LIN {X 0.001,Y -352.403,Z 1885.595,A 0.000,B 0.000,C 90.000,E1 287.166} C_DIS
LIN {X -0.016,Y -356.539,Z 1885.590,A 0.000,B 0.000,C 90.000,E1 286.260} C_DIS
LIN {X -0.091,Y -360.124,Z 1885.585,A 0.000,B 0.000,C 90.000,E1 285.371} C_DIS
LIN {X -0.135,Y -363.075,Z 1885.580,A 0.000,B 0.000,C 90.000,E1 284.481} C_DIS
LIN {X -0.125,Y -364.654,Z 1885.577,A 0.000,B 0.000,C 90.000,E1 283.883} C_DIS
LIN {X -0.190,Y -365.903,Z 1885.574,A 0.000,B 0.000,C 90.000,E1 283.300} C_DIS
LIN {X 0.194,Y -366.725,Z 1885.570,A 0.000,B 0.000,C 90.000,E1 282.647} C_DIS
LIN {X 0.148,Y -367.195,Z 1885.567,A 0.000,B 0.000,C 90.000,E1 282.063} C_DIS
LIN {X 0.107,Y -367.233,Z 1885.564,A 0.000,B 0.000,C 90.000,E1 281.478} C_DIS
LIN {X 0.069,Y -366.898,Z 1885.561,A 0.000,B 0.000,C 90.000,E1 280.894} C_DIS
LIN {X 0.032,Y -366.222,Z 1885.557,A 0.000,B 0.000,C 90.000,E1 280.310} C_DIS
LIN {X -0.009,Y -365.133,Z 1885.554,A 0.000,B 0.000,C 90.000,E1 279.726} C_DIS
LIN {X -0.115,Y -363.688,Z 1885.551,A 0.000,B 0.000,C 90.000,E1 279.151} C_DIS
LIN {X -0.167,Y -361.942,Z 1885.547,A 0.000,B 0.000,C 90.000,E1 278.568} C_DIS
LIN {X 0.040,Y -358.752,Z 1885.542,A 0.000,B 0.000,C 90.000,E1 277.644} C_DIS
LIN {X -0.139,Y -354.719,Z 1885.537,A 0.000,B 0.000,C 90.000,E1 276.777} C_DIS
LIN {X 0.059,Y -351.476,Z 1885.534,A 0.000,B 0.000,C 90.000,E1 276.144} C_DIS
LIN {X -0.111,Y -347.742,Z 1885.531,A 0.000,B 0.000,C 90.000,E1 275.568} C_DIS
LIN {X 0.045,Y -343.441,Z 1885.527,A 0.000,B 0.000,C 90.000,E1 274.935} C_DIS
LIN {X -0.165,Y -338.448,Z 1885.524,A 0.000,B 0.000,C 90.000,E1 274.359} C_DIS
LIN {X -0.059,Y -332.829,Z 1885.521,A 0.000,B 0.000,C 90.000,E1 273.726} C_DIS
LIN {X -0.066,Y -326.939,Z 1885.517,A 0.000,B 0.000,C 90.000,E1 273.154} C_DIS
LIN {X 0.124,Y -320.558,Z 1885.514,A 0.000,B 0.000,C 90.000,E1 272.579} C_DIS
LIN {X 0.017,Y -314.110,Z 1885.512,A 0.000,B 0.000,C 90.000,E1 272.121} C_DIS
LIN {X -0.084,Y -307.356,Z 1885.509,A 0.000,B 0.000,C 90.000,E1 271.718} C_DIS
LIN {X -0.136,Y -300.498,Z 1885.507,A 0.000,B 0.000,C 90.000,E1 271.375} C_DIS
LIN {X 0.073,Y -292.946,Z 1885.506,A 0.000,B 0.000,C 90.000,E1 271.031} C_DIS
LIN {X 0.051,Y -285.090,Z 1885.505,A 0.000,B 0.000,C 90.000,E1 270.802} C_DIS
LIN {X -0.071,Y -273.586,Z 1885.503,A 0.000,B 0.000,C 90.000,E1 270.573} C_DIS
LIN {X 0.101,Y -252.260,Z 1885.501,A 0.000,B 0.000,C 90.000,E1 270.115} C_DIS
LIN {X -0.047,Y -240.338,Z 1885.500,A 0.000,B 0.000,C 90.000,E1 269.943} C_DIS
LIN {X -0.106,Y -228.165,Z 1885.499,A 0.000,B 0.000,C 90.000,E1 269.828} C_DIS
LIN {X 0.098,Y -226.995,Z 1885.499,A 0.000,B 0.000,C 90.000,E1 269.771} C_DIS
LIN {X 0.059,Y -181.515,Z 1885.499,A 0.000,B 0.000,C 90.000,E1 269.771} C_DIS
LIN {X 0.072,Y -180.907,Z 1885.475,A 0.000,B 0.000,C 90.000,E1 265.469} C_DIS
LIN {X -0.050,Y -180.746,Z 1885.470,A 0.000,B 0.000,C 90.000,E1 264.666} C_DIS
LIN {X 0.017,Y -178.838,Z 1885.442,A 0.000,B 0.000,C 90.000,E1 259.577} C_DIS
LIN {X -0.085,Y -175.882,Z 1885.414,A 0.000,B 0.000,C 90.000,E1 254.519} C_DIS
LIN {X 0.021,Y -174.545,Z 1885.404,A 0.000,B 0.000,C 90.000,E1 252.779} C_DIS
LIN {X -0.046,Y -171.530,Z 1885.381,A 0.000,B 0.000,C 90.000,E1 248.518} C_DIS
LIN {X -0.053,Y -167.755,Z 1885.357,A 0.000,B 0.000,C 90.000,E1 244.204} C_DIS
LIN {X 0.037,Y -166.460,Z 1885.347,A 0.000,B 0.000,C 90.000,E1 242.436} C_DIS
LIN {X 0.026,Y -163.175,Z 1885.328,A 0.000,B 0.000,C 90.000,E1 238.948} C_DIS
LIN {X 0.075,Y -161.135,Z 1885.313,A 0.000,B 0.000,C 90.000,E1 236.294} C_DIS
LIN {X -0.023,Y -157.156,Z 1885.288,A 0.000,B 0.000,C 90.000,E1 231.904} C_DIS
LIN {X 0.001,Y -155.888,Z 1885.278,A 0.000,B 0.000,C 90.000,E1 230.114} C_DIS
LIN {X -0.041,Y -152.138,Z 1885.254,A 0.000,B 0.000,C 90.000,E1 225.648} C_DIS
LIN {X -0.021,Y -150.388,Z 1885.239,A 0.000,B 0.000,C 90.000,E1 222.933} C_DIS
LIN {X 0.003,Y -147.119,Z 1885.213,A 0.000,B 0.000,C 90.000,E1 218.382} C_DIS
LIN {X -0.005,Y -145.684,Z 1885.198,A 0.000,B 0.000,C 90.000,E1 215.644} C_DIS
LIN {X -0.008,Y -143.065,Z 1885.172,A 0.000,B 0.000,C 90.000,E1 211.052} C_DIS
LIN {X 0.050,Y -141.687,Z 1885.152,A 0.000,B 0.000,C 90.000,E1 207.334} C_DIS
LIN {X -0.022,Y -139.459,Z 1885.116,A 0.000,B 0.000,C 90.000,E1 200.865} C_DIS
LIN {X 0.079,Y -139.194,Z 1885.105,A 0.000,B 0.000,C 90.000,E1 198.960} C_DIS
LIN {X -0.035,Y -138.324,Z 1885.054,A 0.000,B 0.000,C 90.000,E1 189.670} C_DIS
LIN {X -0.030,Y -139.452,Z 1885.007,A 0.000,B 0.000,C 90.000,E1 181.260} C_DIS
LIN {X 0.050,Y -140.998,Z 1884.976,A 0.000,B 0.000,C 90.000,E1 175.641} C_DIS
LIN {X -0.001,Y -142.753,Z 1884.955,A 0.000,B 0.000,C 90.000,E1 171.951} C_DIS
LIN {X -0.044,Y -145.153,Z 1884.930,A 0.000,B 0.000,C 90.000,E1 167.353} C_DIS
LIN {X -0.052,Y -147.776,Z 1884.909,A 0.000,B 0.000,C 90.000,E1 163.685} C_DIS
LIN {X 0.028,Y -150.453,Z 1884.889,A 0.000,B 0.000,C 90.000,E1 160.007} C_DIS
LIN {X -0.038,Y -153.902,Z 1884.869,A 0.000,B 0.000,C 90.000,E1 156.410} C_DIS
LIN {X 0.028,Y -157.313,Z 1884.849,A 0.000,B 0.000,C 90.000,E1 152.794} C_DIS
LIN {X -0.026,Y -161.500,Z 1884.829,A 0.000,B 0.000,C 90.000,E1 149.253} C_DIS
LIN {X -0.010,Y -165.699,Z 1884.810,A 0.000,B 0.000,C 90.000,E1 145.722} C_DIS
LIN {X 0.116,Y -170.643,Z 1884.790,A 0.000,B 0.000,C 90.000,E1 142.190} C_DIS
LIN {X 0.028,Y -175.519,Z 1884.771,A 0.000,B 0.000,C 90.000,E1 138.771} C_DIS
LIN {X 0.023,Y -181.139,Z 1884.752,A 0.000,B 0.000,C 90.000,E1 135.364} C_DIS
LIN {X 0.021,Y -186.590,Z 1884.733,A 0.000,B 0.000,C 90.000,E1 132.000} C_DIS
LIN {X 0.091,Y -191.201,Z 1884.719,A 0.000,B 0.000,C 90.000,E1 129.483} C_DIS
LIN {X 0.015,Y -197.011,Z 1884.701,A 0.000,B 0.000,C 90.000,E1 126.217} C_DIS
LIN {X -0.066,Y -200.281,Z 1884.692,A 0.000,B 0.000,C 90.000,E1 124.612} C_DIS
LIN {X -0.073,Y -207.773,Z 1884.670,A 0.000,B 0.000,C 90.000,E1 120.590} C_DIS
LIN {X 0.113,Y -210.945,Z 1884.661,A 0.000,B 0.000,C 90.000,E1 118.949} C_DIS
LIN {X -0.066,Y -216.817,Z 1884.644,A 0.000,B 0.000,C 90.000,E1 115.848} C_DIS
LIN {X 0.083,Y -218.433,Z 1884.639,A 0.000,B 0.000,C 90.000,E1 115.027} C_DIS
LIN {X -0.079,Y -221.158,Z 1884.630,A 0.000,B 0.000,C 90.000,E1 113.515} C_DIS
LIN {X -0.007,Y -224.115,Z 1884.621,A 0.000,B 0.000,C 90.000,E1 111.844} C_DIS
LIN {X -0.044,Y -283.396,Z 1884.621,A 0.000,B 0.000,C 90.000,E1 111.844} C_DIS
LIN {X 0.060,Y -286.175,Z 1884.621,A 0.000,B 0.000,C 90.000,E1 111.770} C_DIS
LIN {X 0.099,Y -291.202,Z 1884.619,A 0.000,B 0.000,C 90.000,E1 111.461} C_DIS
LIN {X 0.032,Y -293.997,Z 1884.618,A 0.000,B 0.000,C 90.000,E1 111.173} C_DIS
LIN {X 0.068,Y -296.048,Z 1884.616,A 0.000,B 0.000,C 90.000,E1 110.865} C_DIS
LIN {X -0.046,Y -309.093,Z 1884.603,A 0.000,B 0.000,C 90.000,E1 108.598} C_DIS
LIN {X 0.047,Y -323.638,Z 1884.591,A 0.000,B 0.000,C 90.000,E1 106.315} C_DIS
LIN {X 0.008,Y -337.287,Z 1884.580,A 0.000,B 0.000,C 90.000,E1 104.426} C_DIS
LIN {X -0.102,Y -352.119,Z 1884.570,A 0.000,B 0.000,C 90.000,E1 102.591} C_DIS
LIN {X -0.120,Y -370.511,Z 1884.558,A 0.000,B 0.000,C 90.000,E1 100.546} C_DIS
LIN {X -0.077,Y -389.326,Z 1884.548,A 0.000,B 0.000,C 90.000,E1 98.681} C_DIS
LIN {X 0.195,Y -408.561,Z 1884.539,A 0.000,B 0.000,C 90.000,E1 96.947} C_DIS
LIN {X -0.005,Y -430.922,Z 1884.529,A 0.000,B 0.000,C 90.000,E1 95.220} C_DIS
LIN {X 0.152,Y -439.357,Z 1884.526,A 0.000,B 0.000,C 90.000,E1 94.588} C_DIS
LIN {X -0.073,Y -441.584,Z 1884.525,A 0.000,B 0.000,C 90.000,E1 94.416} C_DIS
LIN {X -0.138,Y -443.567,Z 1884.523,A 0.000,B 0.000,C 90.000,E1 94.188} C_DIS
LIN {X -0.172,Y -445.091,Z 1884.522,A 0.000,B 0.000,C 90.000,E1 93.955} C_DIS
LIN {X 0.007,Y -446.387,Z 1884.520,A 0.000,B 0.000,C 90.000,E1 93.669} C_DIS
LIN {X 0.188,Y -447.352,Z 1884.519,A 0.000,B 0.000,C 90.000,E1 93.383} C_DIS
LIN {X 0.146,Y -448.456,Z 1884.516,A 0.000,B 0.000,C 90.000,E1 92.865} C_DIS
LIN {X 0.086,Y -448.602,Z 1884.513,A 0.000,B 0.000,C 90.000,E1 92.350} C_DIS
LIN {X 0.037,Y -447.816,Z 1884.510,A 0.000,B 0.000,C 90.000,E1 91.835} C_DIS
LIN {X 0.000,Y -445.975,Z 1884.507,A 0.000,B 0.000,C 90.000,E1 91.318} C_DIS
LIN {X -0.053,Y -442.903,Z 1884.504,A 0.000,B 0.000,C 90.000,E1 90.802} C_DIS
LIN {X -0.162,Y -431.386,Z 1884.494,A 0.000,B 0.000,C 90.000,E1 88.969} C_DIS
LIN {X -0.184,Y -421.317,Z 1884.485,A 0.000,B 0.000,C 90.000,E1 87.364} C_DIS
LIN {X 0.139,Y -409.543,Z 1884.475,A 0.000,B 0.000,C 90.000,E1 85.412} C_DIS
LIN {X -0.166,Y -397.645,Z 1884.464,A 0.000,B 0.000,C 90.000,E1 83.514} C_DIS
LIN {X 0.167,Y -385.682,Z 1884.453,A 0.000,B 0.000,C 90.000,E1 81.489} C_DIS
LIN {X -0.072,Y -373.809,Z 1884.442,A 0.000,B 0.000,C 90.000,E1 79.511} C_DIS
LIN {X 0.188,Y -355.793,Z 1884.424,A 0.000,B 0.000,C 90.000,E1 76.228} C_DIS
LIN {X -0.142,Y -341.985,Z 1884.409,A 0.000,B 0.000,C 90.000,E1 73.559} C_DIS
LIN {X 0.129,Y -330.104,Z 1884.395,A 0.000,B 0.000,C 90.000,E1 71.040} C_DIS
LIN {X -0.057,Y -317.077,Z 1884.379,A 0.000,B 0.000,C 90.000,E1 68.230} C_DIS
LIN {X 0.046,Y -304.672,Z 1884.363,A 0.000,B 0.000,C 90.000,E1 65.305} C_DIS
LIN {X 0.048,Y -295.143,Z 1884.350,A 0.000,B 0.000,C 90.000,E1 62.999} C_DIS
LIN {X -0.020,Y -285.826,Z 1884.337,A 0.000,B 0.000,C 90.000,E1 60.667} C_DIS
LIN {X -0.010,Y -276.398,Z 1884.324,A 0.000,B 0.000,C 90.000,E1 58.280} C_DIS
LIN {X -0.150,Y -266.915,Z 1884.310,A 0.000,B 0.000,C 90.000,E1 55.881} C_DIS
LIN {X 0.025,Y -257.306,Z 1884.297,A 0.000,B 0.000,C 90.000,E1 53.371} C_DIS
LIN {X -0.120,Y -247.700,Z 1884.283,A 0.000,B 0.000,C 90.000,E1 50.884} C_DIS
LIN {X -0.146,Y -238.217,Z 1884.268,A 0.000,B 0.000,C 90.000,E1 48.324} C_DIS
LIN {X -0.021,Y -226.401,Z 1884.250,A 0.000,B 0.000,C 90.000,E1 44.919} C_DIS
LIN {X -0.055,Y -215.186,Z 1884.230,A 0.000,B 0.000,C 90.000,E1 41.472} C_DIS
LIN {X 0.051,Y -205.981,Z 1884.213,A 0.000,B 0.000,C 90.000,E1 38.302} C_DIS
LIN {X 0.048,Y -197.685,Z 1884.195,A 0.000,B 0.000,C 90.000,E1 35.105} C_DIS
LIN {X -0.042,Y -190.108,Z 1884.177,A 0.000,B 0.000,C 90.000,E1 31.878} C_DIS
LIN {X -0.025,Y -183.281,Z 1884.159,A 0.000,B 0.000,C 90.000,E1 28.565} C_DIS
LIN {X -0.031,Y -177.125,Z 1884.140,A 0.000,B 0.000,C 90.000,E1 25.207} C_DIS
LIN {X 0.063,Y -171.807,Z 1884.121,A 0.000,B 0.000,C 90.000,E1 21.770} C_DIS
LIN {X -0.061,Y -167.257,Z 1884.102,A 0.000,B 0.000,C 90.000,E1 18.362} C_DIS
LIN {X 0.082,Y -163.533,Z 1884.083,A 0.000,B 0.000,C 90.000,E1 14.828} C_DIS
LIN {X -0.087,Y -159.741,Z 1884.058,A 0.000,B 0.000,C 90.000,E1 10.489} C_DIS
LIN {X -0.023,Y -157.111,Z 1884.033,A 0.000,B 0.000,C 90.000,E1 6.030} C_DIS
LIN {X 0.000,Y -154.819,Z 1884.000,A 0.000,B 0.000,C 90.000,E1 360.000} C_DIS
LIN {X -0.016,Y -154.068,Z 1883.948,A 0.000,B 0.000,C 90.000,E1 350.557} C_DIS
LIN {X -0.014,Y -156.089,Z 1883.908,A 0.000,B 0.000,C 90.000,E1 343.378} C_DIS
LIN {X 0.017,Y -158.516,Z 1883.883,A 0.000,B 0.000,C 90.000,E1 338.901} C_DIS
LIN {X 0.031,Y -162.145,Z 1883.858,A 0.000,B 0.000,C 90.000,E1 334.460} C_DIS
LIN {X 0.082,Y -166.114,Z 1883.839,A 0.000,B 0.000,C 90.000,E1 330.923} C_DIS
LIN {X 0.014,Y -169.717,Z 1883.824,A 0.000,B 0.000,C 90.000,E1 328.329} C_DIS
LIN {X 0.051,Y -173.031,Z 1883.812,A 0.000,B 0.000,C 90.000,E1 326.215} C_DIS
LIN {X 0.035,Y -182.366,Z 1883.812,A 0.000,B 0.000,C 90.000,E1 326.215} C_DIS
LIN {X 0.053,Y -185.804,Z 1883.810,A 0.000,B 0.000,C 90.000,E1 325.722} C_DIS
LIN {X 0.055,Y -188.638,Z 1883.805,A 0.000,B 0.000,C 90.000,E1 324.895} C_DIS
LIN {X 0.040,Y -190.835,Z 1883.800,A 0.000,B 0.000,C 90.000,E1 324.069} C_DIS
LIN {X -0.001,Y -194.525,Z 1883.791,A 0.000,B 0.000,C 90.000,E1 322.431} C_DIS
LIN {X -0.036,Y -199.322,Z 1883.778,A 0.000,B 0.000,C 90.000,E1 319.989} C_DIS
LIN {X -0.086,Y -206.996,Z 1883.755,A 0.000,B 0.000,C 90.000,E1 315.972} C_DIS
LIN {X 0.014,Y -210.390,Z 1883.746,A 0.000,B 0.000,C 90.000,E1 314.352} C_DIS
LIN {X 0.054,Y -215.246,Z 1883.735,A 0.000,B 0.000,C 90.000,E1 312.366} C_DIS
LIN {X -0.029,Y -219.816,Z 1883.727,A 0.000,B 0.000,C 90.000,E1 310.825} C_DIS
LIN {X -0.028,Y -225.338,Z 1883.718,A 0.000,B 0.000,C 90.000,E1 309.277} C_DIS
LIN {X -0.008,Y -233.096,Z 1883.708,A 0.000,B 0.000,C 90.000,E1 307.363} C_DIS
LIN {X -0.148,Y -246.896,Z 1883.691,A 0.000,B 0.000,C 90.000,E1 304.405} C_DIS
LIN {X -0.004,Y -256.206,Z 1883.681,A 0.000,B 0.000,C 90.000,E1 302.546} C_DIS
LIN {X 0.129,Y -272.970,Z 1883.665,A 0.000,B 0.000,C 90.000,E1 299.667} C_DIS
LIN {X 0.053,Y -290.803,Z 1883.650,A 0.000,B 0.000,C 90.000,E1 296.924} C_DIS
LIN {X 0.128,Y -304.184,Z 1883.638,A 0.000,B 0.000,C 90.000,E1 294.899} C_DIS
LIN {X 0.139,Y -315.278,Z 1883.629,A 0.000,B 0.000,C 90.000,E1 293.259} C_DIS
LIN {X 0.084,Y -326.017,Z 1883.620,A 0.000,B 0.000,C 90.000,E1 291.663} C_DIS
LIN {X -0.088,Y -334.306,Z 1883.613,A 0.000,B 0.000,C 90.000,E1 290.429} C_DIS
LIN {X 0.162,Y -340.187,Z 1883.608,A 0.000,B 0.000,C 90.000,E1 289.450} C_DIS
LIN {X 0.040,Y -345.657,Z 1883.603,A 0.000,B 0.000,C 90.000,E1 288.544} C_DIS
LIN {X -0.039,Y -350.699,Z 1883.598,A 0.000,B 0.000,C 90.000,E1 287.638} C_DIS
LIN {X -0.068,Y -355.164,Z 1883.593,A 0.000,B 0.000,C 90.000,E1 286.732} C_DIS
LIN {X -0.163,Y -358.994,Z 1883.588,A 0.000,B 0.000,C 90.000,E1 285.843} C_DIS
LIN {X 0.177,Y -361.272,Z 1883.585,A 0.000,B 0.000,C 90.000,E1 285.190} C_DIS
LIN {X 0.184,Y -363.238,Z 1883.581,A 0.000,B 0.000,C 90.000,E1 284.592} C_DIS
LIN {X 0.106,Y -364.874,Z 1883.578,A 0.000,B 0.000,C 90.000,E1 284.008} C_DIS
LIN {X 0.129,Y -366.174,Z 1883.575,A 0.000,B 0.000,C 90.000,E1 283.411} C_DIS
LIN {X 0.075,Y -367.127,Z 1883.571,A 0.000,B 0.000,C 90.000,E1 282.827} C_DIS
LIN {X 0.031,Y -367.638,Z 1883.568,A 0.000,B 0.000,C 90.000,E1 282.243} C_DIS
LIN {X -0.006,Y -367.773,Z 1883.565,A 0.000,B 0.000,C 90.000,E1 281.658} C_DIS
LIN {X -0.039,Y -367.520,Z 1883.562,A 0.000,B 0.000,C 90.000,E1 281.074} C_DIS
LIN {X -0.071,Y -366.899,Z 1883.558,A 0.000,B 0.000,C 90.000,E1 280.489} C_DIS
LIN {X -0.107,Y -365.890,Z 1883.555,A 0.000,B 0.000,C 90.000,E1 279.905} C_DIS
LIN {X -0.148,Y -364.512,Z 1883.552,A 0.000,B 0.000,C 90.000,E1 279.321} C_DIS
LIN {X 0.107,Y -362.801,Z 1883.548,A 0.000,B 0.000,C 90.000,E1 278.690} C_DIS
LIN {X 0.015,Y -359.690,Z 1883.543,A 0.000,B 0.000,C 90.000,E1 277.814} C_DIS
LIN {X -0.112,Y -357.204,Z 1883.540,A 0.000,B 0.000,C 90.000,E1 277.239} C_DIS
LIN {X 0.046,Y -352.729,Z 1883.535,A 0.000,B 0.000,C 90.000,E1 276.315} C_DIS
LIN {X -0.119,Y -349.129,Z 1883.532,A 0.000,B 0.000,C 90.000,E1 275.739} C_DIS
LIN {X 0.045,Y -344.915,Z 1883.528,A 0.000,B 0.000,C 90.000,E1 275.106} C_DIS
LIN {X -0.158,Y -340.117,Z 1883.525,A 0.000,B 0.000,C 90.000,E1 274.531} C_DIS
LIN {X -0.050,Y -334.635,Z 1883.522,A 0.000,B 0.000,C 90.000,E1 273.898} C_DIS
LIN {X -0.021,Y -325.851,Z 1883.517,A 0.000,B 0.000,C 90.000,E1 273.037} C_DIS
LIN {X -0.020,Y -319.652,Z 1883.514,A 0.000,B 0.000,C 90.000,E1 272.522} C_DIS
LIN {X -0.061,Y -313.156,Z 1883.511,A 0.000,B 0.000,C 90.000,E1 272.064} C_DIS
LIN {X -0.089,Y -306.393,Z 1883.509,A 0.000,B 0.000,C 90.000,E1 271.661} C_DIS
LIN {X -0.103,Y -299.365,Z 1883.507,A 0.000,B 0.000,C 90.000,E1 271.318} C_DIS
LIN {X -0.102,Y -291.908,Z 1883.506,A 0.000,B 0.000,C 90.000,E1 271.031} C_DIS
LIN {X -0.080,Y -284.020,Z 1883.504,A 0.000,B 0.000,C 90.000,E1 270.802} C_DIS
LIN {X 0.003,Y -268.400,Z 1883.503,A 0.000,B 0.000,C 90.000,E1 270.458} C_DIS
LIN {X -0.028,Y -250.496,Z 1883.501,A 0.000,B 0.000,C 90.000,E1 270.115} C_DIS
LIN {X 0.097,Y -238.266,Z 1883.500,A 0.000,B 0.000,C 90.000,E1 269.885} C_DIS
LIN {X -0.098,Y -227.892,Z 1883.499,A 0.000,B 0.000,C 90.000,E1 269.828} C_DIS
LIN {X 0.101,Y -225.810,Z 1883.499,A 0.000,B 0.000,C 90.000,E1 269.771} C_DIS
LIN {X 0.059,Y -181.515,Z 1883.499,A 0.000,B 0.000,C 90.000,E1 269.771} C_DIS
LIN {X -0.011,Y -180.907,Z 1883.475,A 0.000,B 0.000,C 90.000,E1 265.527} C_DIS
LIN {X 0.046,Y -180.760,Z 1883.470,A 0.000,B 0.000,C 90.000,E1 264.666} C_DIS
LIN {X -0.062,Y -178.853,Z 1883.442,A 0.000,B 0.000,C 90.000,E1 259.634} C_DIS
LIN {X 0.010,Y -175.896,Z 1883.414,A 0.000,B 0.000,C 90.000,E1 254.519} C_DIS
LIN {X -0.051,Y -174.572,Z 1883.405,A 0.000,B 0.000,C 90.000,E1 252.834} C_DIS
LIN {X -0.015,Y -171.555,Z 1883.381,A 0.000,B 0.000,C 90.000,E1 248.539} C_DIS
LIN {X 0.040,Y -167.779,Z 1883.357,A 0.000,B 0.000,C 90.000,E1 244.204} C_DIS
LIN {X -0.019,Y -166.491,Z 1883.347,A 0.000,B 0.000,C 90.000,E1 242.487} C_DIS
LIN {X -0.023,Y -163.202,Z 1883.328,A 0.000,B 0.000,C 90.000,E1 238.997} C_DIS
LIN {X 0.032,Y -161.165,Z 1883.313,A 0.000,B 0.000,C 90.000,E1 236.342} C_DIS
LIN {X 0.067,Y -157.181,Z 1883.288,A 0.000,B 0.000,C 90.000,E1 231.904} C_DIS
LIN {X -0.010,Y -155.911,Z 1883.279,A 0.000,B 0.000,C 90.000,E1 230.150} C_DIS
LIN {X 0.046,Y -152.161,Z 1883.254,A 0.000,B 0.000,C 90.000,E1 225.648} C_DIS
LIN {X 0.066,Y -150.410,Z 1883.239,A 0.000,B 0.000,C 90.000,E1 222.933} C_DIS
LIN {X 0.089,Y -147.140,Z 1883.213,A 0.000,B 0.000,C 90.000,E1 218.382} C_DIS
LIN {X -0.005,Y -145.699,Z 1883.198,A 0.000,B 0.000,C 90.000,E1 215.678} C_DIS
LIN {X 0.003,Y -143.082,Z 1883.173,A 0.000,B 0.000,C 90.000,E1 211.082} C_DIS
LIN {X 0.008,Y -141.700,Z 1883.152,A 0.000,B 0.000,C 90.000,E1 207.385} C_DIS
LIN {X -0.070,Y -139.466,Z 1883.116,A 0.000,B 0.000,C 90.000,E1 200.918} C_DIS
LIN {X -0.016,Y -139.199,Z 1883.106,A 0.000,B 0.000,C 90.000,E1 199.033} C_DIS
LIN {X 0.048,Y -138.327,Z 1883.054,A 0.000,B 0.000,C 90.000,E1 189.670} C_DIS
LIN {X 0.053,Y -139.446,Z 1883.007,A 0.000,B 0.000,C 90.000,E1 181.260} C_DIS
LIN {X -0.007,Y -140.985,Z 1882.976,A 0.000,B 0.000,C 90.000,E1 175.698} C_DIS
LIN {X -0.057,Y -142.739,Z 1882.955,A 0.000,B 0.000,C 90.000,E1 172.008} C_DIS
LIN {X 0.041,Y -145.132,Z 1882.930,A 0.000,B 0.000,C 90.000,E1 167.353} C_DIS
LIN {X 0.035,Y -147.755,Z 1882.909,A 0.000,B 0.000,C 90.000,E1 163.685} C_DIS
LIN {X -0.026,Y -150.426,Z 1882.889,A 0.000,B 0.000,C 90.000,E1 160.061} C_DIS
LIN {X -0.011,Y -153.868,Z 1882.869,A 0.000,B 0.000,C 90.000,E1 156.433} C_DIS
LIN {X 0.045,Y -157.278,Z 1882.849,A 0.000,B 0.000,C 90.000,E1 152.820} C_DIS
LIN {X -0.017,Y -161.458,Z 1882.829,A 0.000,B 0.000,C 90.000,E1 149.282} C_DIS
LIN {X -0.012,Y -165.658,Z 1882.810,A 0.000,B 0.000,C 90.000,E1 145.754} C_DIS
LIN {X -0.030,Y -170.593,Z 1882.790,A 0.000,B 0.000,C 90.000,E1 142.271} C_DIS
LIN {X 0.009,Y -175.471,Z 1882.771,A 0.000,B 0.000,C 90.000,E1 138.809} C_DIS
LIN {X -0.008,Y -181.093,Z 1882.752,A 0.000,B 0.000,C 90.000,E1 135.405} C_DIS
LIN {X -0.019,Y -186.536,Z 1882.734,A 0.000,B 0.000,C 90.000,E1 132.043} C_DIS
LIN {X -0.077,Y -191.152,Z 1882.720,A 0.000,B 0.000,C 90.000,E1 129.564} C_DIS
LIN {X 0.001,Y -196.954,Z 1882.701,A 0.000,B 0.000,C 90.000,E1 126.251} C_DIS
LIN {X 0.037,Y -200.220,Z 1882.692,A 0.000,B 0.000,C 90.000,E1 124.612} C_DIS
LIN {X 0.032,Y -207.713,Z 1882.670,A 0.000,B 0.000,C 90.000,E1 120.590} C_DIS
LIN {X 0.035,Y -210.896,Z 1882.661,A 0.000,B 0.000,C 90.000,E1 118.999} C_DIS
LIN {X 0.042,Y -216.759,Z 1882.644,A 0.000,B 0.000,C 90.000,E1 115.848} C_DIS
LIN {X 0.062,Y -219.816,Z 1882.635,A 0.000,B 0.000,C 90.000,E1 114.283} C_DIS
LIN {X -0.004,Y -224.113,Z 1882.621,A 0.000,B 0.000,C 90.000,E1 111.844} C_DIS
LIN {X -0.039,Y -283.450,Z 1882.621,A 0.000,B 0.000,C 90.000,E1 111.844} C_DIS
LIN {X -0.173,Y -285.240,Z 1882.621,A 0.000,B 0.000,C 90.000,E1 111.844} C_DIS
LIN {X -0.137,Y -290.888,Z 1882.620,A 0.000,B 0.000,C 90.000,E1 111.535} C_DIS
LIN {X -0.098,Y -293.778,Z 1882.618,A 0.000,B 0.000,C 90.000,E1 111.227} C_DIS
LIN {X -0.023,Y -295.831,Z 1882.616,A 0.000,B 0.000,C 90.000,E1 110.918} C_DIS
LIN {X -0.015,Y -310.819,Z 1882.602,A 0.000,B 0.000,C 90.000,E1 108.308} C_DIS
LIN {X 0.121,Y -325.548,Z 1882.589,A 0.000,B 0.000,C 90.000,E1 106.024} C_DIS
LIN {X -0.120,Y -339.365,Z 1882.579,A 0.000,B 0.000,C 90.000,E1 104.175} C_DIS
LIN {X 0.063,Y -354.377,Z 1882.568,A 0.000,B 0.000,C 90.000,E1 102.299} C_DIS
LIN {X -0.140,Y -372.807,Z 1882.557,A 0.000,B 0.000,C 90.000,E1 100.310} C_DIS
LIN {X -0.037,Y -391.710,Z 1882.547,A 0.000,B 0.000,C 90.000,E1 98.454} C_DIS
LIN {X -0.002,Y -410.953,Z 1882.538,A 0.000,B 0.000,C 90.000,E1 96.777} C_DIS
LIN {X -0.063,Y -433.357,Z 1882.528,A 0.000,B 0.000,C 90.000,E1 95.049} C_DIS
LIN {X -0.085,Y -439.009,Z 1882.526,A 0.000,B 0.000,C 90.000,E1 94.645} C_DIS
LIN {X 0.126,Y -441.326,Z 1882.525,A 0.000,B 0.000,C 90.000,E1 94.416} C_DIS
LIN {X 0.121,Y -444.864,Z 1882.522,A 0.000,B 0.000,C 90.000,E1 93.955} C_DIS
LIN {X -0.151,Y -446.217,Z 1882.521,A 0.000,B 0.000,C 90.000,E1 93.726} C_DIS
LIN {X 0.023,Y -447.225,Z 1882.519,A 0.000,B 0.000,C 90.000,E1 93.440} C_DIS
LIN {X -0.021,Y -448.399,Z 1882.516,A 0.000,B 0.000,C 90.000,E1 92.922} C_DIS
LIN {X -0.081,Y -448.608,Z 1882.513,A 0.000,B 0.000,C 90.000,E1 92.407} C_DIS
LIN {X -0.131,Y -447.885,Z 1882.510,A 0.000,B 0.000,C 90.000,E1 91.892} C_DIS
LIN {X -0.167,Y -446.123,Z 1882.508,A 0.000,B 0.000,C 90.000,E1 91.375} C_DIS
LIN {X 0.029,Y -444.756,Z 1882.506,A 0.000,B 0.000,C 90.000,E1 91.088} C_DIS
LIN {X 0.112,Y -431.590,Z 1882.494,A 0.000,B 0.000,C 90.000,E1 88.969} C_DIS
LIN {X 0.088,Y -421.529,Z 1882.485,A 0.000,B 0.000,C 90.000,E1 87.364} C_DIS
LIN {X 0.000,Y -409.754,Z 1882.475,A 0.000,B 0.000,C 90.000,E1 85.469} C_DIS
LIN {X 0.099,Y -397.859,Z 1882.464,A 0.000,B 0.000,C 90.000,E1 83.514} C_DIS
LIN {X 0.047,Y -385.896,Z 1882.453,A 0.000,B 0.000,C 90.000,E1 81.546} C_DIS
LIN {X 0.186,Y -374.023,Z 1882.442,A 0.000,B 0.000,C 90.000,E1 79.511} C_DIS
LIN {X 0.010,Y -355.989,Z 1882.424,A 0.000,B 0.000,C 90.000,E1 76.297} C_DIS
LIN {X 0.106,Y -342.170,Z 1882.409,A 0.000,B 0.000,C 90.000,E1 73.559} C_DIS
LIN {X 0.060,Y -330.283,Z 1882.395,A 0.000,B 0.000,C 90.000,E1 71.094} C_DIS
LIN {X -0.112,Y -317.246,Z 1882.379,A 0.000,B 0.000,C 90.000,E1 68.284} C_DIS
LIN {X 0.002,Y -304.832,Z 1882.363,A 0.000,B 0.000,C 90.000,E1 65.357} C_DIS
LIN {X 0.015,Y -295.301,Z 1882.350,A 0.000,B 0.000,C 90.000,E1 63.050} C_DIS
LIN {X -0.044,Y -285.982,Z 1882.337,A 0.000,B 0.000,C 90.000,E1 60.717} C_DIS
LIN {X -0.024,Y -276.555,Z 1882.324,A 0.000,B 0.000,C 90.000,E1 58.329} C_DIS
LIN {X 0.068,Y -267.075,Z 1882.311,A 0.000,B 0.000,C 90.000,E1 55.881} C_DIS
LIN {X 0.032,Y -257.469,Z 1882.297,A 0.000,B 0.000,C 90.000,E1 53.417} C_DIS
LIN {X 0.089,Y -247.864,Z 1882.283,A 0.000,B 0.000,C 90.000,E1 50.884} C_DIS
LIN {X 0.058,Y -238.379,Z 1882.269,A 0.000,B 0.000,C 90.000,E1 48.324} C_DIS
LIN {X 0.017,Y -226.553,Z 1882.250,A 0.000,B 0.000,C 90.000,E1 44.960} C_DIS
LIN {X -0.023,Y -215.328,Z 1882.231,A 0.000,B 0.000,C 90.000,E1 41.515} C_DIS
LIN {X -0.051,Y -206.113,Z 1882.213,A 0.000,B 0.000,C 90.000,E1 38.382} C_DIS
LIN {X -0.044,Y -197.803,Z 1882.195,A 0.000,B 0.000,C 90.000,E1 35.185} C_DIS
LIN {X -0.025,Y -190.218,Z 1882.177,A 0.000,B 0.000,C 90.000,E1 31.926} C_DIS
LIN {X -0.011,Y -183.382,Z 1882.159,A 0.000,B 0.000,C 90.000,E1 28.615} C_DIS
LIN {X -0.095,Y -177.212,Z 1882.140,A 0.000,B 0.000,C 90.000,E1 25.283} C_DIS
LIN {X 0.008,Y -171.882,Z 1882.121,A 0.000,B 0.000,C 90.000,E1 21.844} C_DIS
LIN {X -0.053,Y -167.320,Z 1882.102,A 0.000,B 0.000,C 90.000,E1 18.417} C_DIS
LIN {X 0.045,Y -163.582,Z 1882.083,A 0.000,B 0.000,C 90.000,E1 14.898} C_DIS
LIN {X -0.083,Y -159.776,Z 1882.058,A 0.000,B 0.000,C 90.000,E1 10.546} C_DIS
LIN {X -0.019,Y -157.130,Z 1882.034,A 0.000,B 0.000,C 90.000,E1 6.087} C_DIS
LIN {X 0.000,Y -154.811,Z 1882.000,A 0.000,B 0.000,C 90.000,E1 360.000} C_DIS
LIN {X -0.016,Y -154.061,Z 1881.948,A 0.000,B 0.000,C 90.000,E1 350.557} C_DIS
LIN {X -0.015,Y -156.085,Z 1881.908,A 0.000,B 0.000,C 90.000,E1 343.378} C_DIS
LIN {X 0.018,Y -158.514,Z 1881.883,A 0.000,B 0.000,C 90.000,E1 338.901} C_DIS
LIN {X 0.029,Y -162.146,Z 1881.858,A 0.000,B 0.000,C 90.000,E1 334.460} C_DIS
LIN {X 0.081,Y -166.117,Z 1881.839,A 0.000,B 0.000,C 90.000,E1 330.923} C_DIS
LIN {X 0.016,Y -167.691,Z 1881.832,A 0.000,B 0.000,C 90.000,E1 329.744} C_DIS
LIN {X -0.005,Y -179.393,Z 1881.832,A 0.000,B 0.000,C 90.000,E1 329.744} C_DIS
LIN {X -0.069,Y -180.709,Z 1881.831,A 0.000,B 0.000,C 90.000,E1 329.665} C_DIS
LIN {X 0.001,Y -183.016,Z 1881.829,A 0.000,B 0.000,C 90.000,E1 329.203} C_DIS
LIN {X 0.106,Y -185.737,Z 1881.824,A 0.000,B 0.000,C 90.000,E1 328.329} C_DIS
LIN {X -0.025,Y -187.838,Z 1881.820,A 0.000,B 0.000,C 90.000,E1 327.533} C_DIS
LIN {X -0.044,Y -189.706,Z 1881.815,A 0.000,B 0.000,C 90.000,E1 326.707} C_DIS
LIN {X -0.057,Y -192.993,Z 1881.806,A 0.000,B 0.000,C 90.000,E1 325.055} C_DIS
LIN {X 0.069,Y -197.354,Z 1881.792,A 0.000,B 0.000,C 90.000,E1 322.557} C_DIS
LIN {X -0.035,Y -201.413,Z 1881.779,A 0.000,B 0.000,C 90.000,E1 320.150} C_DIS
LIN {X -0.025,Y -208.318,Z 1881.756,A 0.000,B 0.000,C 90.000,E1 316.134} C_DIS
LIN {X 0.092,Y -211.448,Z 1881.747,A 0.000,B 0.000,C 90.000,E1 314.514} C_DIS
LIN {X 0.106,Y -215.017,Z 1881.739,A 0.000,B 0.000,C 90.000,E1 312.933} C_DIS
LIN {X 0.014,Y -219.110,Z 1881.730,A 0.000,B 0.000,C 90.000,E1 311.391} C_DIS
LIN {X -0.084,Y -222.769,Z 1881.724,A 0.000,B 0.000,C 90.000,E1 310.253} C_DIS
LIN {X 0.038,Y -229.801,Z 1881.713,A 0.000,B 0.000,C 90.000,E1 308.302} C_DIS
LIN {X 0.146,Y -239.338,Z 1881.700,A 0.000,B 0.000,C 90.000,E1 306.011} C_DIS
LIN {X -0.041,Y -249.819,Z 1881.688,A 0.000,B 0.000,C 90.000,E1 303.833} C_DIS
LIN {X 0.131,Y -257.449,Z 1881.680,A 0.000,B 0.000,C 90.000,E1 302.339} C_DIS
LIN {X 0.102,Y -276.603,Z 1881.662,A 0.000,B 0.000,C 90.000,E1 299.155} C_DIS
LIN {X 0.141,Y -292.312,Z 1881.649,A 0.000,B 0.000,C 90.000,E1 296.744} C_DIS
LIN {X -0.022,Y -305.724,Z 1881.638,A 0.000,B 0.000,C 90.000,E1 294.771} C_DIS
LIN {X 0.015,Y -316.828,Z 1881.629,A 0.000,B 0.000,C 90.000,E1 293.131} C_DIS
LIN {X -0.029,Y -327.589,Z 1881.620,A 0.000,B 0.000,C 90.000,E1 291.535} C_DIS
LIN {X 0.130,Y -335.881,Z 1881.613,A 0.000,B 0.000,C 90.000,E1 290.248} C_DIS
LIN {X -0.039,Y -343.557,Z 1881.606,A 0.000,B 0.000,C 90.000,E1 289.033} C_DIS
LIN {X -0.118,Y -350.475,Z 1881.599,A 0.000,B 0.000,C 90.000,E1 287.819} C_DIS
LIN {X -0.150,Y -355.067,Z 1881.594,A 0.000,B 0.000,C 90.000,E1 286.913} C_DIS
LIN {X 0.098,Y -359.015,Z 1881.589,A 0.000,B 0.000,C 90.000,E1 285.969} C_DIS
LIN {X 0.144,Y -362.375,Z 1881.584,A 0.000,B 0.000,C 90.000,E1 285.064} C_DIS
LIN {X 0.029,Y -365.090,Z 1881.579,A 0.000,B 0.000,C 90.000,E1 284.189} C_DIS
LIN {X 0.054,Y -366.463,Z 1881.576,A 0.000,B 0.000,C 90.000,E1 283.592} C_DIS
LIN {X 0.002,Y -367.481,Z 1881.572,A 0.000,B 0.000,C 90.000,E1 283.008} C_DIS
LIN {X 0.040,Y -368.097,Z 1881.569,A 0.000,B 0.000,C 90.000,E1 282.411} C_DIS
LIN {X 0.002,Y -368.304,Z 1881.566,A 0.000,B 0.000,C 90.000,E1 281.827} C_DIS
LIN {X -0.030,Y -368.129,Z 1881.562,A 0.000,B 0.000,C 90.000,E1 281.243} C_DIS
LIN {X -0.062,Y -367.557,Z 1881.559,A 0.000,B 0.000,C 90.000,E1 280.658} C_DIS
LIN {X -0.095,Y -366.596,Z 1881.556,A 0.000,B 0.000,C 90.000,E1 280.074} C_DIS
LIN {X -0.193,Y -365.309,Z 1881.553,A 0.000,B 0.000,C 90.000,E1 279.500} C_DIS
LIN {X 0.124,Y -363.681,Z 1881.549,A 0.000,B 0.000,C 90.000,E1 278.859} C_DIS
LIN {X -0.013,Y -360.664,Z 1881.544,A 0.000,B 0.000,C 90.000,E1 277.992} C_DIS
LIN {X -0.086,Y -358.278,Z 1881.541,A 0.000,B 0.000,C 90.000,E1 277.409} C_DIS
LIN {X 0.079,Y -353.919,Z 1881.536,A 0.000,B 0.000,C 90.000,E1 276.486} C_DIS
LIN {X -0.081,Y -350.467,Z 1881.533,A 0.000,B 0.000,C 90.000,E1 275.910} C_DIS
LIN {X 0.089,Y -346.487,Z 1881.529,A 0.000,B 0.000,C 90.000,E1 275.277} C_DIS
LIN {X -0.107,Y -341.833,Z 1881.526,A 0.000,B 0.000,C 90.000,E1 274.702} C_DIS
LIN {X -0.014,Y -336.494,Z 1881.523,A 0.000,B 0.000,C 90.000,E1 274.073} C_DIS
LIN {X -0.131,Y -330.650,Z 1881.519,A 0.000,B 0.000,C 90.000,E1 273.498} C_DIS
LIN {X 0.045,Y -324.814,Z 1881.516,A 0.000,B 0.000,C 90.000,E1 272.922} C_DIS
LIN {X 0.054,Y -318.434,Z 1881.513,A 0.000,B 0.000,C 90.000,E1 272.407} C_DIS
LIN {X 0.060,Y -311.792,Z 1881.511,A 0.000,B 0.000,C 90.000,E1 271.949} C_DIS
LIN {X 0.080,Y -304.838,Z 1881.509,A 0.000,B 0.000,C 90.000,E1 271.547} C_DIS
LIN {X 0.118,Y -297.634,Z 1881.507,A 0.000,B 0.000,C 90.000,E1 271.203} C_DIS
LIN {X -0.093,Y -290.034,Z 1881.505,A 0.000,B 0.000,C 90.000,E1 270.974} C_DIS
LIN {X 0.010,Y -282.390,Z 1881.504,A 0.000,B 0.000,C 90.000,E1 270.745} C_DIS
LIN {X 0.000,Y -256.706,Z 1881.501,A 0.000,B 0.000,C 90.000,E1 270.229} C_DIS
LIN {X 0.052,Y -241.282,Z 1881.500,A 0.000,B 0.000,C 90.000,E1 269.943} C_DIS
LIN {X 0.016,Y -230.701,Z 1881.499,A 0.000,B 0.000,C 90.000,E1 269.828} C_DIS
LIN {X -0.099,Y -225.098,Z 1881.499,A 0.000,B 0.000,C 90.000,E1 269.828} C_DIS
LIN {X 0.079,Y -181.517,Z 1881.499,A 0.000,B 0.000,C 90.000,E1 269.771} C_DIS
LIN {X -0.022,Y -180.899,Z 1881.474,A 0.000,B 0.000,C 90.000,E1 265.241} C_DIS
LIN {X -0.072,Y -180.214,Z 1881.464,A 0.000,B 0.000,C 90.000,E1 263.571} C_DIS
LIN {X 0.058,Y -179.034,Z 1881.445,A 0.000,B 0.000,C 90.000,E1 260.151} C_DIS
LIN {X -0.057,Y -178.690,Z 1881.441,A 0.000,B 0.000,C 90.000,E1 259.342} C_DIS
LIN {X 0.054,Y -175.740,Z 1881.412,A 0.000,B 0.000,C 90.000,E1 254.212} C_DIS
LIN {X 0.050,Y -171.923,Z 1881.384,A 0.000,B 0.000,C 90.000,E1 249.082} C_DIS
LIN {X 0.024,Y -171.297,Z 1881.379,A 0.000,B 0.000,C 90.000,E1 248.230} C_DIS
LIN {X 0.070,Y -167.559,Z 1881.355,A 0.000,B 0.000,C 90.000,E1 243.896} C_DIS
LIN {X 0.084,Y -166.185,Z 1881.345,A 0.000,B 0.000,C 90.000,E1 242.153} C_DIS
LIN {X 0.073,Y -162.955,Z 1881.326,A 0.000,B 0.000,C 90.000,E1 238.663} C_DIS
LIN {X -0.103,Y -160.863,Z 1881.311,A 0.000,B 0.000,C 90.000,E1 236.087} C_DIS
LIN {X 0.097,Y -157.637,Z 1881.292,A 0.000,B 0.000,C 90.000,E1 232.477} C_DIS
LIN {X 0.034,Y -155.675,Z 1881.277,A 0.000,B 0.000,C 90.000,E1 229.828} C_DIS
LIN {X 0.086,Y -151.942,Z 1881.252,A 0.000,B 0.000,C 90.000,E1 225.324} C_DIS
LIN {X 0.102,Y -150.180,Z 1881.237,A 0.000,B 0.000,C 90.000,E1 222.609} C_DIS
LIN {X 0.020,Y -146.954,Z 1881.212,A 0.000,B 0.000,C 90.000,E1 218.096} C_DIS
LIN {X 0.008,Y -145.541,Z 1881.196,A 0.000,B 0.000,C 90.000,E1 215.358} C_DIS
LIN {X -0.075,Y -142.937,Z 1881.171,A 0.000,B 0.000,C 90.000,E1 210.797} C_DIS
LIN {X -0.018,Y -141.562,Z 1881.150,A 0.000,B 0.000,C 90.000,E1 207.078} C_DIS
LIN {X 0.034,Y -139.409,Z 1881.114,A 0.000,B 0.000,C 90.000,E1 200.556} C_DIS
LIN {X -0.043,Y -139.130,Z 1881.104,A 0.000,B 0.000,C 90.000,E1 198.725} C_DIS
LIN {X -0.016,Y -138.350,Z 1881.057,A 0.000,B 0.000,C 90.000,E1 190.310} C_DIS
LIN {X -0.029,Y -139.498,Z 1881.005,A 0.000,B 0.000,C 90.000,E1 180.974} C_DIS
LIN {X 0.052,Y -141.119,Z 1880.974,A 0.000,B 0.000,C 90.000,E1 175.355} C_DIS
LIN {X 0.005,Y -142.499,Z 1880.959,A 0.000,B 0.000,C 90.000,E1 172.591} C_DIS
LIN {X -0.048,Y -144.754,Z 1880.933,A 0.000,B 0.000,C 90.000,E1 167.993} C_DIS
LIN {X 0.043,Y -147.363,Z 1880.913,A 0.000,B 0.000,C 90.000,E1 164.283} C_DIS
LIN {X -0.035,Y -150.690,Z 1880.887,A 0.000,B 0.000,C 90.000,E1 159.752} C_DIS
LIN {X 0.048,Y -154.170,Z 1880.867,A 0.000,B 0.000,C 90.000,E1 156.102} C_DIS
LIN {X -0.021,Y -157.603,Z 1880.847,A 0.000,B 0.000,C 90.000,E1 152.538} C_DIS
LIN {X -0.071,Y -161.855,Z 1880.828,A 0.000,B 0.000,C 90.000,E1 148.997} C_DIS
LIN {X -0.054,Y -166.047,Z 1880.808,A 0.000,B 0.000,C 90.000,E1 145.468} C_DIS
LIN {X -0.062,Y -171.050,Z 1880.789,A 0.000,B 0.000,C 90.000,E1 141.984} C_DIS
LIN {X -0.033,Y -175.922,Z 1880.770,A 0.000,B 0.000,C 90.000,E1 138.528} C_DIS
LIN {X -0.040,Y -180.160,Z 1880.755,A 0.000,B 0.000,C 90.000,E1 135.972} C_DIS
LIN {X -0.072,Y -185.578,Z 1880.737,A 0.000,B 0.000,C 90.000,E1 132.609} C_DIS
LIN {X -0.022,Y -190.167,Z 1880.723,A 0.000,B 0.000,C 90.000,E1 130.092} C_DIS
LIN {X 0.024,Y -197.497,Z 1880.700,A 0.000,B 0.000,C 90.000,E1 125.964} C_DIS
LIN {X 0.065,Y -200.766,Z 1880.691,A 0.000,B 0.000,C 90.000,E1 124.326} C_DIS
LIN {X -0.024,Y -206.656,Z 1880.673,A 0.000,B 0.000,C 90.000,E1 121.131} C_DIS
LIN {X -0.033,Y -209.953,Z 1880.664,A 0.000,B 0.000,C 90.000,E1 119.539} C_DIS
LIN {X -0.004,Y -217.307,Z 1880.642,A 0.000,B 0.000,C 90.000,E1 115.591} C_DIS
LIN {X -0.051,Y -218.930,Z 1880.638,A 0.000,B 0.000,C 90.000,E1 114.823} C_DIS
LIN {X -0.002,Y -224.111,Z 1880.621,A 0.000,B 0.000,C 90.000,E1 111.844} C_DIS
LIN {X -0.054,Y -283.977,Z 1880.621,A 0.000,B 0.000,C 90.000,E1 111.844} C_DIS
LIN {X -0.016,Y -287.865,Z 1880.621,A 0.000,B 0.000,C 90.000,E1 111.716} C_DIS
LIN {X -0.094,Y -290.801,Z 1880.620,A 0.000,B 0.000,C 90.000,E1 111.535} C_DIS
LIN {X 0.061,Y -294.515,Z 1880.617,A 0.000,B 0.000,C 90.000,E1 111.099} C_DIS
LIN {X 0.098,Y -298.118,Z 1880.614,A 0.000,B 0.000,C 90.000,E1 110.482} C_DIS
LIN {X 0.046,Y -311.529,Z 1880.601,A 0.000,B 0.000,C 90.000,E1 108.181} C_DIS
LIN {X -0.118,Y -326.331,Z 1880.589,A 0.000,B 0.000,C 90.000,E1 105.953} C_DIS
LIN {X -0.115,Y -340.214,Z 1880.578,A 0.000,B 0.000,C 90.000,E1 104.064} C_DIS
LIN {X 0.091,Y -355.300,Z 1880.568,A 0.000,B 0.000,C 90.000,E1 102.187} C_DIS
LIN {X -0.042,Y -373.755,Z 1880.557,A 0.000,B 0.000,C 90.000,E1 100.197} C_DIS
LIN {X 0.132,Y -392.678,Z 1880.546,A 0.000,B 0.000,C 90.000,E1 98.341} C_DIS
LIN {X -0.175,Y -411.938,Z 1880.537,A 0.000,B 0.000,C 90.000,E1 96.720} C_DIS
LIN {X -0.185,Y -434.360,Z 1880.528,A 0.000,B 0.000,C 90.000,E1 94.992} C_DIS
LIN {X -0.194,Y -439.910,Z 1880.525,A 0.000,B 0.000,C 90.000,E1 94.588} C_DIS
LIN {X 0.023,Y -441.988,Z 1880.524,A 0.000,B 0.000,C 90.000,E1 94.359} C_DIS
LIN {X -0.123,Y -443.940,Z 1880.523,A 0.000,B 0.000,C 90.000,E1 94.131} C_DIS
LIN {X 0.206,Y -445.431,Z 1880.521,A 0.000,B 0.000,C 90.000,E1 93.841} C_DIS
LIN {X -0.059,Y -446.636,Z 1880.520,A 0.000,B 0.000,C 90.000,E1 93.612} C_DIS
LIN {X 0.124,Y -447.523,Z 1880.519,A 0.000,B 0.000,C 90.000,E1 93.326} C_DIS
LIN {X 0.084,Y -448.499,Z 1880.516,A 0.000,B 0.000,C 90.000,E1 92.808} C_DIS
LIN {X 0.025,Y -448.527,Z 1880.513,A 0.000,B 0.000,C 90.000,E1 92.293} C_DIS
LIN {X -0.010,Y -447.616,Z 1880.510,A 0.000,B 0.000,C 90.000,E1 91.776} C_DIS
LIN {X -0.060,Y -445.621,Z 1880.507,A 0.000,B 0.000,C 90.000,E1 91.260} C_DIS
LIN {X -0.187,Y -439.152,Z 1880.501,A 0.000,B 0.000,C 90.000,E1 90.229} C_DIS
LIN {X 0.060,Y -427.614,Z 1880.491,A 0.000,B 0.000,C 90.000,E1 88.339} C_DIS
LIN {X 0.184,Y -414.145,Z 1880.479,A 0.000,B 0.000,C 90.000,E1 86.159} C_DIS
LIN {X -0.025,Y -402.300,Z 1880.468,A 0.000,B 0.000,C 90.000,E1 84.261} C_DIS
LIN {X -0.035,Y -390.337,Z 1880.457,A 0.000,B 0.000,C 90.000,E1 82.299} C_DIS
LIN {X 0.141,Y -378.425,Z 1880.446,A 0.000,B 0.000,C 90.000,E1 80.274} C_DIS
LIN {X 0.128,Y -361.741,Z 1880.430,A 0.000,B 0.000,C 90.000,E1 77.353} C_DIS
LIN {X -0.120,Y -346.097,Z 1880.413,A 0.000,B 0.000,C 90.000,E1 74.393} C_DIS
LIN {X -0.165,Y -334.107,Z 1880.400,A 0.000,B 0.000,C 90.000,E1 71.945} C_DIS
LIN {X 0.118,Y -322.396,Z 1880.386,A 0.000,B 0.000,C 90.000,E1 69.390} C_DIS
LIN {X -0.039,Y -309.734,Z 1880.370,A 0.000,B 0.000,C 90.000,E1 66.538} C_DIS
LIN {X -0.176,Y -300.207,Z 1880.357,A 0.000,B 0.000,C 90.000,E1 64.280} C_DIS
LIN {X -0.028,Y -288.111,Z 1880.340,A 0.000,B 0.000,C 90.000,E1 61.257} C_DIS
LIN {X 0.033,Y -278.709,Z 1880.327,A 0.000,B 0.000,C 90.000,E1 58.869} C_DIS
LIN {X 0.172,Y -269.223,Z 1880.314,A 0.000,B 0.000,C 90.000,E1 56.421} C_DIS
LIN {X -0.025,Y -261.028,Z 1880.302,A 0.000,B 0.000,C 90.000,E1 54.356} C_DIS
LIN {X 0.114,Y -251.429,Z 1880.288,A 0.000,B 0.000,C 90.000,E1 51.823} C_DIS
LIN {X 0.003,Y -241.866,Z 1880.274,A 0.000,B 0.000,C 90.000,E1 49.299} C_DIS
LIN {X 0.121,Y -231.189,Z 1880.257,A 0.000,B 0.000,C 90.000,E1 46.296} C_DIS
LIN {X -0.041,Y -220.959,Z 1880.240,A 0.000,B 0.000,C 90.000,E1 43.299} C_DIS
LIN {X 0.045,Y -211.307,Z 1880.223,A 0.000,B 0.000,C 90.000,E1 40.172} C_DIS
LIN {X -0.091,Y -203.521,Z 1880.208,A 0.000,B 0.000,C 90.000,E1 37.443} C_DIS
LIN {X 0.022,Y -195.439,Z 1880.190,A 0.000,B 0.000,C 90.000,E1 34.199} C_DIS
LIN {X 0.036,Y -188.083,Z 1880.172,A 0.000,B 0.000,C 90.000,E1 30.924} C_DIS
LIN {X 0.068,Y -181.449,Z 1880.153,A 0.000,B 0.000,C 90.000,E1 27.590} C_DIS
LIN {X -0.063,Y -175.524,Z 1880.135,A 0.000,B 0.000,C 90.000,E1 24.259} C_DIS
LIN {X 0.085,Y -170.434,Z 1880.116,A 0.000,B 0.000,C 90.000,E1 20.791} C_DIS
LIN {X 0.037,Y -166.118,Z 1880.096,A 0.000,B 0.000,C 90.000,E1 17.347} C_DIS
LIN {X -0.051,Y -162.589,Z 1880.077,A 0.000,B 0.000,C 90.000,E1 13.883} C_DIS
LIN {X 0.039,Y -159.030,Z 1880.052,A 0.000,B 0.000,C 90.000,E1 9.443} C_DIS
LIN {X -0.024,Y -156.259,Z 1880.023,A 0.000,B 0.000,C 90.000,E1 4.131} C_DIS
LIN {X -0.016,Y -154.131,Z 1879.982,A 0.000,B 0.000,C 90.000,E1 356.846} C_DIS
LIN {X -0.002,Y -155.107,Z 1879.923,A 0.000,B 0.000,C 90.000,E1 346.061} C_DIS
LIN {X 0.034,Y -157.414,Z 1879.893,A 0.000,B 0.000,C 90.000,E1 340.678} C_DIS
LIN {X 0.031,Y -160.560,Z 1879.868,A 0.000,B 0.000,C 90.000,E1 336.230} C_DIS
LIN {X 0.007,Y -163.398,Z 1879.851,A 0.000,B 0.000,C 90.000,E1 333.256} C_DIS
LIN {X -0.014,Y -176.524,Z 1879.851,A 0.000,B 0.000,C 90.000,E1 333.256} C_DIS
LIN {X 0.014,Y -177.708,Z 1879.851,A 0.000,B 0.000,C 90.000,E1 333.179} C_DIS
LIN {X -0.006,Y -178.543,Z 1879.850,A 0.000,B 0.000,C 90.000,E1 333.076} C_DIS
LIN {X 0.046,Y -180.286,Z 1879.848,A 0.000,B 0.000,C 90.000,E1 332.692} C_DIS
LIN {X 0.041,Y -182.965,Z 1879.844,A 0.000,B 0.000,C 90.000,E1 331.847} C_DIS
LIN {X 0.054,Y -185.022,Z 1879.839,A 0.000,B 0.000,C 90.000,E1 331.001} C_DIS
LIN {X -0.080,Y -186.828,Z 1879.834,A 0.000,B 0.000,C 90.000,E1 330.205} C_DIS
LIN {X -0.069,Y -189.977,Z 1879.825,A 0.000,B 0.000,C 90.000,E1 328.535} C_DIS
LIN {X 0.099,Y -194.148,Z 1879.811,A 0.000,B 0.000,C 90.000,E1 326.008} C_DIS
LIN {X 0.020,Y -197.985,Z 1879.798,A 0.000,B 0.000,C 90.000,E1 323.577} C_DIS
LIN {X -0.046,Y -202.854,Z 1879.780,A 0.000,B 0.000,C 90.000,E1 320.356} C_DIS
LIN {X 0.012,Y -209.198,Z 1879.757,A 0.000,B 0.000,C 90.000,E1 316.338} C_DIS
LIN {X 0.076,Y -213.727,Z 1879.744,A 0.000,B 0.000,C 90.000,E1 313.947} C_DIS
LIN {X 0.023,Y -218.271,Z 1879.733,A 0.000,B 0.000,C 90.000,E1 312.000} C_DIS
LIN {X 0.056,Y -221.486,Z 1879.727,A 0.000,B 0.000,C 90.000,E1 310.825} C_DIS
LIN {X 0.080,Y -226.594,Z 1879.718,A 0.000,B 0.000,C 90.000,E1 309.277} C_DIS
LIN {X -0.014,Y -233.783,Z 1879.708,A 0.000,B 0.000,C 90.000,E1 307.397} C_DIS
LIN {X -0.002,Y -241.877,Z 1879.697,A 0.000,B 0.000,C 90.000,E1 305.518} C_DIS
LIN {X 0.064,Y -252.679,Z 1879.685,A 0.000,B 0.000,C 90.000,E1 303.293} C_DIS
LIN {X -0.079,Y -260.606,Z 1879.677,A 0.000,B 0.000,C 90.000,E1 301.878} C_DIS
LIN {X 0.035,Y -277.880,Z 1879.661,A 0.000,B 0.000,C 90.000,E1 299.027} C_DIS
LIN {X 0.108,Y -293.663,Z 1879.648,A 0.000,B 0.000,C 90.000,E1 296.616} C_DIS
LIN {X -0.032,Y -307.091,Z 1879.637,A 0.000,B 0.000,C 90.000,E1 294.643} C_DIS
LIN {X -0.106,Y -318.202,Z 1879.628,A 0.000,B 0.000,C 90.000,E1 293.025} C_DIS
LIN {X 0.002,Y -329.003,Z 1879.619,A 0.000,B 0.000,C 90.000,E1 291.408} C_DIS
LIN {X 0.178,Y -337.288,Z 1879.612,A 0.000,B 0.000,C 90.000,E1 290.120} C_DIS
LIN {X 0.024,Y -343.053,Z 1879.607,A 0.000,B 0.000,C 90.000,E1 289.214} C_DIS
LIN {X -0.071,Y -348.423,Z 1879.602,A 0.000,B 0.000,C 90.000,E1 288.308} C_DIS
LIN {X -0.124,Y -353.332,Z 1879.597,A 0.000,B 0.000,C 90.000,E1 287.402} C_DIS
LIN {X -0.129,Y -357.623,Z 1879.592,A 0.000,B 0.000,C 90.000,E1 286.496} C_DIS
LIN {X -0.201,Y -361.300,Z 1879.587,A 0.000,B 0.000,C 90.000,E1 285.607} C_DIS
LIN {X 0.156,Y -363.409,Z 1879.583,A 0.000,B 0.000,C 90.000,E1 284.954} C_DIS
LIN {X 0.176,Y -365.220,Z 1879.580,A 0.000,B 0.000,C 90.000,E1 284.356} C_DIS
LIN {X 0.112,Y -366.685,Z 1879.577,A 0.000,B 0.000,C 90.000,E1 283.772} C_DIS
LIN {X 0.145,Y -367.790,Z 1879.573,A 0.000,B 0.000,C 90.000,E1 283.175} C_DIS
LIN {X 0.102,Y -368.483,Z 1879.570,A 0.000,B 0.000,C 90.000,E1 282.591} C_DIS
LIN {X 0.068,Y -368.797,Z 1879.567,A 0.000,B 0.000,C 90.000,E1 282.007} C_DIS
LIN {X 0.040,Y -368.710,Z 1879.563,A 0.000,B 0.000,C 90.000,E1 281.422} C_DIS
LIN {X 0.012,Y -368.227,Z 1879.560,A 0.000,B 0.000,C 90.000,E1 280.838} C_DIS
LIN {X -0.016,Y -367.369,Z 1879.557,A 0.000,B 0.000,C 90.000,E1 280.254} C_DIS
LIN {X -0.049,Y -366.160,Z 1879.554,A 0.000,B 0.000,C 90.000,E1 279.670} C_DIS
LIN {X -0.146,Y -364.588,Z 1879.550,A 0.000,B 0.000,C 90.000,E1 279.095} C_DIS
LIN {X 0.168,Y -362.710,Z 1879.547,A 0.000,B 0.000,C 90.000,E1 278.454} C_DIS
LIN {X 0.024,Y -359.373,Z 1879.542,A 0.000,B 0.000,C 90.000,E1 277.587} C_DIS
LIN {X -0.148,Y -355.228,Z 1879.537,A 0.000,B 0.000,C 90.000,E1 276.720} C_DIS
LIN {X 0.054,Y -351.931,Z 1879.534,A 0.000,B 0.000,C 90.000,E1 276.087} C_DIS
LIN {X 0.155,Y -345.958,Z 1879.529,A 0.000,B 0.000,C 90.000,E1 275.163} C_DIS
LIN {X -0.045,Y -341.211,Z 1879.525,A 0.000,B 0.000,C 90.000,E1 274.588} C_DIS
LIN {X 0.082,Y -335.775,Z 1879.522,A 0.000,B 0.000,C 90.000,E1 273.955} C_DIS
LIN {X -0.018,Y -329.873,Z 1879.519,A 0.000,B 0.000,C 90.000,E1 273.383} C_DIS
LIN {X 0.120,Y -323.767,Z 1879.516,A 0.000,B 0.000,C 90.000,E1 272.808} C_DIS
LIN {X -0.130,Y -317.346,Z 1879.513,A 0.000,B 0.000,C 90.000,E1 272.350} C_DIS
LIN {X -0.030,Y -310.701,Z 1879.510,A 0.000,B 0.000,C 90.000,E1 271.892} C_DIS
LIN {X 0.092,Y -303.813,Z 1879.508,A 0.000,B 0.000,C 90.000,E1 271.489} C_DIS
LIN {X -0.108,Y -296.558,Z 1879.507,A 0.000,B 0.000,C 90.000,E1 271.203} C_DIS
LIN {X 0.022,Y -288.862,Z 1879.505,A 0.000,B 0.000,C 90.000,E1 270.917} C_DIS
LIN {X -0.120,Y -280.986,Z 1879.504,A 0.000,B 0.000,C 90.000,E1 270.745} C_DIS
LIN {X -0.077,Y -255.567,Z 1879.501,A 0.000,B 0.000,C 90.000,E1 270.229} C_DIS
LIN {X 0.038,Y -244.120,Z 1879.500,A 0.000,B 0.000,C 90.000,E1 270.000} C_DIS
LIN {X 0.076,Y -231.178,Z 1879.499,A 0.000,B 0.000,C 90.000,E1 269.828} C_DIS
LIN {X -0.050,Y -226.966,Z 1879.499,A 0.000,B 0.000,C 90.000,E1 269.828} C_DIS
LIN {X -0.059,Y -181.521,Z 1879.499,A 0.000,B 0.000,C 90.000,E1 269.828} C_DIS
LIN {X -0.059,Y -180.907,Z 1879.475,A 0.000,B 0.000,C 90.000,E1 265.527} C_DIS
LIN {X -0.002,Y -180.753,Z 1879.470,A 0.000,B 0.000,C 90.000,E1 264.666} C_DIS
LIN {X 0.067,Y -178.846,Z 1879.442,A 0.000,B 0.000,C 90.000,E1 259.577} C_DIS
LIN {X -0.038,Y -175.890,Z 1879.414,A 0.000,B 0.000,C 90.000,E1 254.519} C_DIS
LIN {X 0.069,Y -174.559,Z 1879.404,A 0.000,B 0.000,C 90.000,E1 252.779} C_DIS
LIN {X -0.062,Y -171.542,Z 1879.381,A 0.000,B 0.000,C 90.000,E1 248.539} C_DIS
LIN {X -0.006,Y -167.767,Z 1879.357,A 0.000,B 0.000,C 90.000,E1 244.204} C_DIS
LIN {X -0.064,Y -166.476,Z 1879.347,A 0.000,B 0.000,C 90.000,E1 242.487} C_DIS
LIN {X -0.067,Y -163.189,Z 1879.328,A 0.000,B 0.000,C 90.000,E1 238.997} C_DIS
LIN {X -0.012,Y -161.150,Z 1879.313,A 0.000,B 0.000,C 90.000,E1 236.342} C_DIS
LIN {X 0.023,Y -157.168,Z 1879.288,A 0.000,B 0.000,C 90.000,E1 231.904} C_DIS
LIN {X -0.054,Y -155.900,Z 1879.278,A 0.000,B 0.000,C 90.000,E1 230.150} C_DIS
LIN {X 0.003,Y -152.150,Z 1879.254,A 0.000,B 0.000,C 90.000,E1 225.648} C_DIS
LIN {X 0.023,Y -150.399,Z 1879.239,A 0.000,B 0.000,C 90.000,E1 222.933} C_DIS
LIN {X 0.047,Y -147.129,Z 1879.213,A 0.000,B 0.000,C 90.000,E1 218.382} C_DIS
LIN {X 0.037,Y -145.692,Z 1879.198,A 0.000,B 0.000,C 90.000,E1 215.644} C_DIS
LIN {X 0.035,Y -143.074,Z 1879.173,A 0.000,B 0.000,C 90.000,E1 211.052} C_DIS
LIN {X -0.034,Y -141.693,Z 1879.152,A 0.000,B 0.000,C 90.000,E1 207.385} C_DIS
LIN {X 0.020,Y -139.463,Z 1879.116,A 0.000,B 0.000,C 90.000,E1 200.865} C_DIS
LIN {X -0.057,Y -139.196,Z 1879.106,A 0.000,B 0.000,C 90.000,E1 199.033} C_DIS
LIN {X 0.006,Y -138.326,Z 1879.054,A 0.000,B 0.000,C 90.000,E1 189.670} C_DIS
LIN {X 0.012,Y -139.449,Z 1879.007,A 0.000,B 0.000,C 90.000,E1 181.260} C_DIS
LIN {X -0.048,Y -140.992,Z 1878.976,A 0.000,B 0.000,C 90.000,E1 175.698} C_DIS
LIN {X 0.043,Y -142.746,Z 1878.955,A 0.000,B 0.000,C 90.000,E1 171.951} C_DIS
LIN {X -0.001,Y -145.143,Z 1878.930,A 0.000,B 0.000,C 90.000,E1 167.353} C_DIS
LIN {X -0.008,Y -147.766,Z 1878.909,A 0.000,B 0.000,C 90.000,E1 163.685} C_DIS
LIN {X -0.069,Y -150.440,Z 1878.889,A 0.000,B 0.000,C 90.000,E1 160.061} C_DIS
LIN {X 0.007,Y -153.885,Z 1878.869,A 0.000,B 0.000,C 90.000,E1 156.410} C_DIS
LIN {X 0.001,Y -157.295,Z 1878.849,A 0.000,B 0.000,C 90.000,E1 152.820} C_DIS
LIN {X 0.019,Y -161.478,Z 1878.829,A 0.000,B 0.000,C 90.000,E1 149.253} C_DIS
LIN {X 0.036,Y -165.678,Z 1878.810,A 0.000,B 0.000,C 90.000,E1 145.722} C_DIS
LIN {X -0.076,Y -170.618,Z 1878.790,A 0.000,B 0.000,C 90.000,E1 142.271} C_DIS
LIN {X 0.077,Y -175.494,Z 1878.771,A 0.000,B 0.000,C 90.000,E1 138.771} C_DIS
LIN {X -0.057,Y -181.116,Z 1878.752,A 0.000,B 0.000,C 90.000,E1 135.405} C_DIS
LIN {X 0.071,Y -186.563,Z 1878.733,A 0.000,B 0.000,C 90.000,E1 132.000} C_DIS
LIN {X 0.021,Y -191.176,Z 1878.720,A 0.000,B 0.000,C 90.000,E1 129.519} C_DIS
LIN {X 0.067,Y -196.982,Z 1878.701,A 0.000,B 0.000,C 90.000,E1 126.217} C_DIS
LIN {X -0.014,Y -200.250,Z 1878.692,A 0.000,B 0.000,C 90.000,E1 124.612} C_DIS
LIN {X -0.021,Y -207.743,Z 1878.670,A 0.000,B 0.000,C 90.000,E1 120.590} C_DIS
LIN {X -0.018,Y -210.921,Z 1878.661,A 0.000,B 0.000,C 90.000,E1 118.999} C_DIS
LIN {X -0.011,Y -216.788,Z 1878.644,A 0.000,B 0.000,C 90.000,E1 115.848} C_DIS
LIN {X 0.098,Y -219.839,Z 1878.635,A 0.000,B 0.000,C 90.000,E1 114.259} C_DIS
LIN {X -0.006,Y -224.114,Z 1878.621,A 0.000,B 0.000,C 90.000,E1 111.844} C_DIS
LIN {X -0.041,Y -283.855,Z 1878.621,A 0.000,B 0.000,C 90.000,E1 111.844} C_DIS
LIN {X 0.130,Y -285.846,Z 1878.621,A 0.000,B 0.000,C 90.000,E1 111.770} C_DIS
LIN {X 0.065,Y -291.065,Z 1878.619,A 0.000,B 0.000,C 90.000,E1 111.482} C_DIS
LIN {X -0.168,Y -293.893,Z 1878.618,A 0.000,B 0.000,C 90.000,E1 111.227} C_DIS
LIN {X -0.122,Y -295.945,Z 1878.616,A 0.000,B 0.000,C 90.000,E1 110.918} C_DIS
LIN {X -0.044,Y -310.960,Z 1878.602,A 0.000,B 0.000,C 90.000,E1 108.290} C_DIS
LIN {X -0.009,Y -325.703,Z 1878.589,A 0.000,B 0.000,C 90.000,E1 106.024} C_DIS
LIN {X 0.077,Y -339.534,Z 1878.578,A 0.000,B 0.000,C 90.000,E1 104.120} C_DIS
LIN {X -0.072,Y -354.560,Z 1878.568,A 0.000,B 0.000,C 90.000,E1 102.299} C_DIS
LIN {X 0.098,Y -372.995,Z 1878.557,A 0.000,B 0.000,C 90.000,E1 100.254} C_DIS
LIN {X -0.159,Y -391.902,Z 1878.547,A 0.000,B 0.000,C 90.000,E1 98.454} C_DIS
LIN {X -0.119,Y -411.148,Z 1878.538,A 0.000,B 0.000,C 90.000,E1 96.777} C_DIS
LIN {X -0.175,Y -433.556,Z 1878.528,A 0.000,B 0.000,C 90.000,E1 95.049} C_DIS
LIN {X -0.195,Y -439.196,Z 1878.526,A 0.000,B 0.000,C 90.000,E1 94.645} C_DIS
LIN {X 0.016,Y -441.455,Z 1878.525,A 0.000,B 0.000,C 90.000,E1 94.416} C_DIS
LIN {X -0.050,Y -444.973,Z 1878.522,A 0.000,B 0.000,C 90.000,E1 93.955} C_DIS
LIN {X 0.124,Y -446.292,Z 1878.521,A 0.000,B 0.000,C 90.000,E1 93.669} C_DIS
LIN {X -0.148,Y -447.273,Z 1878.519,A 0.000,B 0.000,C 90.000,E1 93.440} C_DIS
LIN {X -0.191,Y -448.400,Z 1878.516,A 0.000,B 0.000,C 90.000,E1 92.922} C_DIS
LIN {X 0.197,Y -448.567,Z 1878.513,A 0.000,B 0.000,C 90.000,E1 92.350} C_DIS
LIN {X 0.146,Y -447.802,Z 1878.510,A 0.000,B 0.000,C 90.000,E1 91.835} C_DIS
LIN {X 0.109,Y -445.988,Z 1878.507,A 0.000,B 0.000,C 90.000,E1 91.318} C_DIS
LIN {X -0.140,Y -444.587,Z 1878.506,A 0.000,B 0.000,C 90.000,E1 91.088} C_DIS
LIN {X -0.056,Y -431.413,Z 1878.494,A 0.000,B 0.000,C 90.000,E1 88.969} C_DIS
LIN {X -0.079,Y -421.350,Z 1878.485,A 0.000,B 0.000,C 90.000,E1 87.364} C_DIS
LIN {X -0.167,Y -409.575,Z 1878.475,A 0.000,B 0.000,C 90.000,E1 85.469} C_DIS
LIN {X -0.067,Y -397.677,Z 1878.464,A 0.000,B 0.000,C 90.000,E1 83.514} C_DIS
LIN {X -0.117,Y -385.716,Z 1878.453,A 0.000,B 0.000,C 90.000,E1 81.546} C_DIS
LIN {X 0.024,Y -373.836,Z 1878.442,A 0.000,B 0.000,C 90.000,E1 79.511} C_DIS
LIN {X -0.067,Y -355.815,Z 1878.424,A 0.000,B 0.000,C 90.000,E1 76.284} C_DIS
LIN {X -0.054,Y -342.002,Z 1878.409,A 0.000,B 0.000,C 90.000,E1 73.559} C_DIS
LIN {X -0.098,Y -330.115,Z 1878.395,A 0.000,B 0.000,C 90.000,E1 71.094} C_DIS
LIN {X 0.026,Y -317.082,Z 1878.379,A 0.000,B 0.000,C 90.000,E1 68.230} C_DIS
LIN {X -0.151,Y -304.672,Z 1878.363,A 0.000,B 0.000,C 90.000,E1 65.357} C_DIS
LIN {X 0.125,Y -295.137,Z 1878.350,A 0.000,B 0.000,C 90.000,E1 62.999} C_DIS
LIN {X 0.054,Y -285.816,Z 1878.337,A 0.000,B 0.000,C 90.000,E1 60.667} C_DIS
LIN {X 0.062,Y -276.392,Z 1878.324,A 0.000,B 0.000,C 90.000,E1 58.280} C_DIS
LIN {X -0.081,Y -266.914,Z 1878.310,A 0.000,B 0.000,C 90.000,E1 55.881} C_DIS
LIN {X -0.114,Y -257.311,Z 1878.297,A 0.000,B 0.000,C 90.000,E1 53.417} C_DIS
LIN {X -0.056,Y -247.703,Z 1878.283,A 0.000,B 0.000,C 90.000,E1 50.884} C_DIS
LIN {X -0.084,Y -238.219,Z 1878.268,A 0.000,B 0.000,C 90.000,E1 48.324} C_DIS
LIN {X 0.037,Y -226.399,Z 1878.250,A 0.000,B 0.000,C 90.000,E1 44.919} C_DIS
LIN {X 0.001,Y -215.182,Z 1878.230,A 0.000,B 0.000,C 90.000,E1 41.472} C_DIS
LIN {X -0.024,Y -205.982,Z 1878.213,A 0.000,B 0.000,C 90.000,E1 38.338} C_DIS
LIN {X 0.100,Y -197.686,Z 1878.195,A 0.000,B 0.000,C 90.000,E1 35.105} C_DIS
LIN {X 0.007,Y -190.114,Z 1878.177,A 0.000,B 0.000,C 90.000,E1 31.878} C_DIS
LIN {X 0.022,Y -183.288,Z 1878.159,A 0.000,B 0.000,C 90.000,E1 28.565} C_DIS
LIN {X 0.015,Y -177.130,Z 1878.140,A 0.000,B 0.000,C 90.000,E1 25.207} C_DIS
LIN {X 0.044,Y -171.811,Z 1878.121,A 0.000,B 0.000,C 90.000,E1 21.791} C_DIS
LIN {X -0.017,Y -167.258,Z 1878.102,A 0.000,B 0.000,C 90.000,E1 18.362} C_DIS
LIN {X -0.033,Y -163.527,Z 1878.083,A 0.000,B 0.000,C 90.000,E1 14.883} C_DIS
LIN {X -0.045,Y -159.729,Z 1878.058,A 0.000,B 0.000,C 90.000,E1 10.489} C_DIS
LIN {X 0.019,Y -157.092,Z 1878.034,A 0.000,B 0.000,C 90.000,E1 6.030} C_DIS
LIN {X 0.000,Y -154.794,Z 1878.000,A 0.000,B 0.000,C 90.000,E1 360.000} C_DIS
LIN {X -0.017,Y -154.049,Z 1877.948,A 0.000,B 0.000,C 90.000,E1 350.557} C_DIS
LIN {X -0.016,Y -156.076,Z 1877.908,A 0.000,B 0.000,C 90.000,E1 343.378} C_DIS
LIN {X 0.015,Y -158.510,Z 1877.883,A 0.000,B 0.000,C 90.000,E1 338.901} C_DIS
LIN {X -0.037,Y -160.108,Z 1877.871,A 0.000,B 0.000,C 90.000,E1 336.794} C_DIS
LIN {X -0.060,Y -174.171,Z 1877.871,A 0.000,B 0.000,C 90.000,E1 336.794} C_DIS
LIN {X -0.023,Y -175.010,Z 1877.871,A 0.000,B 0.000,C 90.000,E1 336.741} C_DIS
LIN {X 0.040,Y -175.925,Z 1877.870,A 0.000,B 0.000,C 90.000,E1 336.613} C_DIS
LIN {X 0.034,Y -177.764,Z 1877.868,A 0.000,B 0.000,C 90.000,E1 336.230} C_DIS
LIN {X -0.068,Y -180.350,Z 1877.863,A 0.000,B 0.000,C 90.000,E1 335.409} C_DIS
LIN {X 0.014,Y -182.348,Z 1877.859,A 0.000,B 0.000,C 90.000,E1 334.537} C_DIS
LIN {X -0.046,Y -185.689,Z 1877.849,A 0.000,B 0.000,C 90.000,E1 332.871} C_DIS
LIN {X 0.024,Y -188.568,Z 1877.840,A 0.000,B 0.000,C 90.000,E1 331.179} C_DIS
LIN {X 0.130,Y -192.439,Z 1877.826,A 0.000,B 0.000,C 90.000,E1 328.663} C_DIS
LIN {X 0.079,Y -196.002,Z 1877.812,A 0.000,B 0.000,C 90.000,E1 326.215} C_DIS
LIN {X 0.037,Y -199.425,Z 1877.799,A 0.000,B 0.000,C 90.000,E1 323.783} C_DIS
LIN {X 0.008,Y -203.877,Z 1877.781,A 0.000,B 0.000,C 90.000,E1 320.561} C_DIS
LIN {X -0.040,Y -209.764,Z 1877.759,A 0.000,B 0.000,C 90.000,E1 316.581} C_DIS
LIN {X 0.034,Y -213.983,Z 1877.746,A 0.000,B 0.000,C 90.000,E1 314.190} C_DIS
LIN {X 0.077,Y -217.328,Z 1877.737,A 0.000,B 0.000,C 90.000,E1 312.609} C_DIS
LIN {X 0.013,Y -221.255,Z 1877.728,A 0.000,B 0.000,C 90.000,E1 311.067} C_DIS
LIN {X 0.035,Y -226.045,Z 1877.720,A 0.000,B 0.000,C 90.000,E1 309.519} C_DIS
LIN {X -0.059,Y -231.509,Z 1877.711,A 0.000,B 0.000,C 90.000,E1 308.016} C_DIS
LIN {X -0.052,Y -237.682,Z 1877.703,A 0.000,B 0.000,C 90.000,E1 306.503} C_DIS
LIN {X -0.071,Y -248.059,Z 1877.690,A 0.000,B 0.000,C 90.000,E1 304.278} C_DIS
LIN {X 0.099,Y -257.573,Z 1877.680,A 0.000,B 0.000,C 90.000,E1 302.418} C_DIS
LIN {X 0.040,Y -274.694,Z 1877.664,A 0.000,B 0.000,C 90.000,E1 299.589} C_DIS
LIN {X -0.134,Y -292.703,Z 1877.649,A 0.000,B 0.000,C 90.000,E1 296.873} C_DIS
LIN {X 0.091,Y -303.929,Z 1877.640,A 0.000,B 0.000,C 90.000,E1 295.155} C_DIS
LIN {X 0.107,Y -315.115,Z 1877.631,A 0.000,B 0.000,C 90.000,E1 293.515} C_DIS
LIN {X 0.164,Y -326.060,Z 1877.622,A 0.000,B 0.000,C 90.000,E1 291.897} C_DIS
LIN {X -0.008,Y -334.599,Z 1877.615,A 0.000,B 0.000,C 90.000,E1 290.663} C_DIS
LIN {X -0.186,Y -340.605,Z 1877.610,A 0.000,B 0.000,C 90.000,E1 289.758} C_DIS
LIN {X 0.024,Y -347.983,Z 1877.603,A 0.000,B 0.000,C 90.000,E1 288.489} C_DIS
LIN {X -0.031,Y -353.015,Z 1877.598,A 0.000,B 0.000,C 90.000,E1 287.583} C_DIS
LIN {X -0.038,Y -357.428,Z 1877.593,A 0.000,B 0.000,C 90.000,E1 286.677} C_DIS
LIN {X -0.110,Y -361.195,Z 1877.588,A 0.000,B 0.000,C 90.000,E1 285.788} C_DIS
LIN {X -0.103,Y -363.383,Z 1877.584,A 0.000,B 0.000,C 90.000,E1 285.190} C_DIS
LIN {X -0.084,Y -365.281,Z 1877.581,A 0.000,B 0.000,C 90.000,E1 284.592} C_DIS
LIN {X -0.151,Y -366.857,Z 1877.578,A 0.000,B 0.000,C 90.000,E1 284.008} C_DIS
LIN {X -0.116,Y -368.051,Z 1877.574,A 0.000,B 0.000,C 90.000,E1 283.411} C_DIS
LIN {X -0.159,Y -368.855,Z 1877.571,A 0.000,B 0.000,C 90.000,E1 282.827} C_DIS
LIN {X -0.192,Y -369.284,Z 1877.568,A 0.000,B 0.000,C 90.000,E1 282.243} C_DIS
LIN {X 0.143,Y -369.267,Z 1877.565,A 0.000,B 0.000,C 90.000,E1 281.602} C_DIS
LIN {X 0.191,Y -368.895,Z 1877.561,A 0.000,B 0.000,C 90.000,E1 281.007} C_DIS
LIN {X 0.097,Y -368.123,Z 1877.558,A 0.000,B 0.000,C 90.000,E1 280.433} C_DIS
LIN {X 0.071,Y -366.975,Z 1877.555,A 0.000,B 0.000,C 90.000,E1 279.849} C_DIS
LIN {X 0.038,Y -365.475,Z 1877.552,A 0.000,B 0.000,C 90.000,E1 279.265} C_DIS
LIN {X -0.005,Y -363.673,Z 1877.548,A 0.000,B 0.000,C 90.000,E1 278.681} C_DIS
LIN {X -0.143,Y -360.453,Z 1877.543,A 0.000,B 0.000,C 90.000,E1 277.814} C_DIS
LIN {X 0.047,Y -356.505,Z 1877.538,A 0.000,B 0.000,C 90.000,E1 276.891} C_DIS
LIN {X -0.098,Y -353.372,Z 1877.535,A 0.000,B 0.000,C 90.000,E1 276.315} C_DIS
LIN {X 0.091,Y -349.665,Z 1877.532,A 0.000,B 0.000,C 90.000,E1 275.682} C_DIS
LIN {X -0.089,Y -345.430,Z 1877.528,A 0.000,B 0.000,C 90.000,E1 275.106} C_DIS
LIN {X 0.052,Y -340.581,Z 1877.525,A 0.000,B 0.000,C 90.000,E1 274.473} C_DIS
LIN {X 0.160,Y -335.036,Z 1877.521,A 0.000,B 0.000,C 90.000,E1 273.841} C_DIS
LIN {X 0.082,Y -329.068,Z 1877.518,A 0.000,B 0.000,C 90.000,E1 273.269} C_DIS
LIN {X 0.001,Y -322.997,Z 1877.515,A 0.000,B 0.000,C 90.000,E1 272.751} C_DIS
LIN {X -0.151,Y -316.607,Z 1877.513,A 0.000,B 0.000,C 90.000,E1 272.293} C_DIS
LIN {X -0.035,Y -309.805,Z 1877.510,A 0.000,B 0.000,C 90.000,E1 271.835} C_DIS
LIN {X 0.125,Y -302.825,Z 1877.508,A 0.000,B 0.000,C 90.000,E1 271.432} C_DIS
LIN {X -0.027,Y -295.320,Z 1877.506,A 0.000,B 0.000,C 90.000,E1 271.146} C_DIS
LIN {X -0.112,Y -287.830,Z 1877.505,A 0.000,B 0.000,C 90.000,E1 270.917} C_DIS
LIN {X -0.015,Y -276.256,Z 1877.504,A 0.000,B 0.000,C 90.000,E1 270.630} C_DIS
LIN {X 0.099,Y -251.342,Z 1877.501,A 0.000,B 0.000,C 90.000,E1 270.115} C_DIS
LIN {X -0.025,Y -238.808,Z 1877.500,A 0.000,B 0.000,C 90.000,E1 269.943} C_DIS
LIN {X 0.073,Y -230.118,Z 1877.499,A 0.000,B 0.000,C 90.000,E1 269.828} C_DIS
LIN {X -0.039,Y -225.058,Z 1877.499,A 0.000,B 0.000,C 90.000,E1 269.828} C_DIS
LIN {X -0.053,Y -181.521,Z 1877.499,A 0.000,B 0.000,C 90.000,E1 269.828} C_DIS
LIN {X 0.077,Y -180.908,Z 1877.475,A 0.000,B 0.000,C 90.000,E1 265.527} C_DIS
LIN {X -0.045,Y -180.770,Z 1877.471,A 0.000,B 0.000,C 90.000,E1 264.723} C_DIS
LIN {X 0.026,Y -178.866,Z 1877.443,A 0.000,B 0.000,C 90.000,E1 259.634} C_DIS
LIN {X -0.073,Y -175.909,Z 1877.414,A 0.000,B 0.000,C 90.000,E1 254.574} C_DIS
LIN {X -0.017,Y -174.595,Z 1877.405,A 0.000,B 0.000,C 90.000,E1 252.851} C_DIS
LIN {X -0.090,Y -171.578,Z 1877.381,A 0.000,B 0.000,C 90.000,E1 248.592} C_DIS
LIN {X 0.052,Y -167.800,Z 1877.357,A 0.000,B 0.000,C 90.000,E1 244.229} C_DIS
LIN {X 0.066,Y -166.518,Z 1877.347,A 0.000,B 0.000,C 90.000,E1 242.487} C_DIS
LIN {X 0.054,Y -162.519,Z 1877.323,A 0.000,B 0.000,C 90.000,E1 238.122} C_DIS
LIN {X 0.025,Y -161.192,Z 1877.313,A 0.000,B 0.000,C 90.000,E1 236.373} C_DIS
LIN {X -0.072,Y -157.203,Z 1877.289,A 0.000,B 0.000,C 90.000,E1 231.984} C_DIS
LIN {X -0.050,Y -155.931,Z 1877.279,A 0.000,B 0.000,C 90.000,E1 230.194} C_DIS
LIN {X -0.089,Y -152.183,Z 1877.254,A 0.000,B 0.000,C 90.000,E1 225.729} C_DIS
LIN {X -0.068,Y -150.430,Z 1877.239,A 0.000,B 0.000,C 90.000,E1 223.014} C_DIS
LIN {X -0.040,Y -147.158,Z 1877.214,A 0.000,B 0.000,C 90.000,E1 218.463} C_DIS
LIN {X -0.073,Y -145.172,Z 1877.193,A 0.000,B 0.000,C 90.000,E1 214.818} C_DIS
LIN {X -0.038,Y -142.322,Z 1877.163,A 0.000,B 0.000,C 90.000,E1 209.283} C_DIS
LIN {X 0.084,Y -141.711,Z 1877.152,A 0.000,B 0.000,C 90.000,E1 207.385} C_DIS
LIN {X 0.006,Y -139.472,Z 1877.116,A 0.000,B 0.000,C 90.000,E1 200.918} C_DIS
LIN {X -0.072,Y -139.204,Z 1877.106,A 0.000,B 0.000,C 90.000,E1 199.087} C_DIS
LIN {X -0.014,Y -138.329,Z 1877.054,A 0.000,B 0.000,C 90.000,E1 189.726} C_DIS
LIN {X -0.011,Y -139.439,Z 1877.007,A 0.000,B 0.000,C 90.000,E1 181.318} C_DIS
LIN {X 0.069,Y -140.972,Z 1876.976,A 0.000,B 0.000,C 90.000,E1 175.698} C_DIS
LIN {X 0.019,Y -142.728,Z 1876.956,A 0.000,B 0.000,C 90.000,E1 172.008} C_DIS
LIN {X -0.024,Y -145.113,Z 1876.930,A 0.000,B 0.000,C 90.000,E1 167.409} C_DIS
LIN {X -0.029,Y -147.737,Z 1876.910,A 0.000,B 0.000,C 90.000,E1 163.740} C_DIS
LIN {X 0.053,Y -150.401,Z 1876.889,A 0.000,B 0.000,C 90.000,E1 160.061} C_DIS
LIN {X -0.072,Y -153.836,Z 1876.869,A 0.000,B 0.000,C 90.000,E1 156.485} C_DIS
LIN {X -0.013,Y -157.247,Z 1876.849,A 0.000,B 0.000,C 90.000,E1 152.871} C_DIS
LIN {X -0.074,Y -161.420,Z 1876.829,A 0.000,B 0.000,C 90.000,E1 149.331} C_DIS
LIN {X -0.064,Y -165.621,Z 1876.810,A 0.000,B 0.000,C 90.000,E1 145.801} C_DIS
LIN {X 0.056,Y -170.550,Z 1876.791,A 0.000,B 0.000,C 90.000,E1 142.271} C_DIS
LIN {X -0.036,Y -175.428,Z 1876.771,A 0.000,B 0.000,C 90.000,E1 138.852} C_DIS
LIN {X 0.081,Y -181.052,Z 1876.752,A 0.000,B 0.000,C 90.000,E1 135.405} C_DIS
LIN {X -0.053,Y -186.487,Z 1876.734,A 0.000,B 0.000,C 90.000,E1 132.081} C_DIS
LIN {X 0.015,Y -191.108,Z 1876.720,A 0.000,B 0.000,C 90.000,E1 129.564} C_DIS
LIN {X -0.064,Y -196.902,Z 1876.702,A 0.000,B 0.000,C 90.000,E1 126.297} C_DIS
LIN {X -0.034,Y -200.163,Z 1876.693,A 0.000,B 0.000,C 90.000,E1 124.659} C_DIS
LIN {X 0.128,Y -207.659,Z 1876.670,A 0.000,B 0.000,C 90.000,E1 120.590} C_DIS
LIN {X 0.030,Y -210.851,Z 1876.661,A 0.000,B 0.000,C 90.000,E1 119.027} C_DIS
LIN {X -0.055,Y -216.707,Z 1876.644,A 0.000,B 0.000,C 90.000,E1 115.899} C_DIS
LIN {X -0.040,Y -219.774,Z 1876.635,A 0.000,B 0.000,C 90.000,E1 114.335} C_DIS
LIN {X 0.016,Y -224.103,Z 1876.621,A 0.000,B 0.000,C 90.000,E1 111.844} C_DIS
LIN {X -0.012,Y -283.289,Z 1876.621,A 0.000,B 0.000,C 90.000,E1 111.844} C_DIS
LIN {X 0.108,Y -288.435,Z 1876.620,A 0.000,B 0.000,C 90.000,E1 111.663} C_DIS
LIN {X -0.007,Y -290.609,Z 1876.620,A 0.000,B 0.000,C 90.000,E1 111.535} C_DIS
LIN {X 0.034,Y -293.580,Z 1876.618,A 0.000,B 0.000,C 90.000,E1 111.227} C_DIS
LIN {X -0.029,Y -297.265,Z 1876.615,A 0.000,B 0.000,C 90.000,E1 110.663} C_DIS
LIN {X -0.121,Y -310.602,Z 1876.602,A 0.000,B 0.000,C 90.000,E1 108.362} C_DIS
LIN {X 0.001,Y -325.309,Z 1876.589,A 0.000,B 0.000,C 90.000,E1 106.079} C_DIS
LIN {X -0.006,Y -339.104,Z 1876.579,A 0.000,B 0.000,C 90.000,E1 104.189} C_DIS
LIN {X -0.083,Y -354.094,Z 1876.569,A 0.000,B 0.000,C 90.000,E1 102.355} C_DIS
LIN {X 0.051,Y -372.519,Z 1876.557,A 0.000,B 0.000,C 90.000,E1 100.310} C_DIS
LIN {X 0.145,Y -391.416,Z 1876.547,A 0.000,B 0.000,C 90.000,E1 98.454} C_DIS
LIN {X 0.172,Y -410.652,Z 1876.538,A 0.000,B 0.000,C 90.000,E1 96.777} C_DIS
LIN {X 0.102,Y -433.051,Z 1876.528,A 0.000,B 0.000,C 90.000,E1 95.049} C_DIS
LIN {X 0.079,Y -438.709,Z 1876.526,A 0.000,B 0.000,C 90.000,E1 94.645} C_DIS
LIN {X -0.151,Y -441.098,Z 1876.525,A 0.000,B 0.000,C 90.000,E1 94.473} C_DIS
LIN {X -0.087,Y -444.657,Z 1876.522,A 0.000,B 0.000,C 90.000,E1 94.012} C_DIS
LIN {X 0.084,Y -446.050,Z 1876.521,A 0.000,B 0.000,C 90.000,E1 93.726} C_DIS
LIN {X -0.189,Y -447.092,Z 1876.519,A 0.000,B 0.000,C 90.000,E1 93.498} C_DIS
LIN {X 0.214,Y -448.320,Z 1876.516,A 0.000,B 0.000,C 90.000,E1 92.922} C_DIS
LIN {X 0.153,Y -448.577,Z 1876.513,A 0.000,B 0.000,C 90.000,E1 92.407} C_DIS
LIN {X 0.101,Y -447.906,Z 1876.511,A 0.000,B 0.000,C 90.000,E1 91.892} C_DIS
LIN {X 0.065,Y -446.205,Z 1876.508,A 0.000,B 0.000,C 90.000,E1 91.375} C_DIS
LIN {X -0.184,Y -444.877,Z 1876.506,A 0.000,B 0.000,C 90.000,E1 91.146} C_DIS
LIN {X -0.093,Y -431.715,Z 1876.495,A 0.000,B 0.000,C 90.000,E1 89.026} C_DIS
LIN {X -0.110,Y -421.662,Z 1876.486,A 0.000,B 0.000,C 90.000,E1 87.421} C_DIS
LIN {X -0.189,Y -409.888,Z 1876.475,A 0.000,B 0.000,C 90.000,E1 85.527} C_DIS
LIN {X -0.080,Y -397.994,Z 1876.464,A 0.000,B 0.000,C 90.000,E1 83.571} C_DIS
LIN {X -0.122,Y -386.032,Z 1876.453,A 0.000,B 0.000,C 90.000,E1 81.602} C_DIS
LIN {X 0.027,Y -374.152,Z 1876.442,A 0.000,B 0.000,C 90.000,E1 79.567} C_DIS
LIN {X -0.134,Y -356.108,Z 1876.424,A 0.000,B 0.000,C 90.000,E1 76.353} C_DIS
LIN {X -0.025,Y -342.277,Z 1876.409,A 0.000,B 0.000,C 90.000,E1 73.614} C_DIS
LIN {X -0.059,Y -330.381,Z 1876.395,A 0.000,B 0.000,C 90.000,E1 71.148} C_DIS
LIN {X 0.131,Y -318.755,Z 1876.381,A 0.000,B 0.000,C 90.000,E1 68.592} C_DIS
LIN {X -0.120,Y -306.280,Z 1876.365,A 0.000,B 0.000,C 90.000,E1 65.741} C_DIS
LIN {X -0.080,Y -296.732,Z 1876.352,A 0.000,B 0.000,C 90.000,E1 63.435} C_DIS
LIN {X 0.132,Y -286.055,Z 1876.338,A 0.000,B 0.000,C 90.000,E1 60.717} C_DIS
LIN {X 0.148,Y -276.629,Z 1876.324,A 0.000,B 0.000,C 90.000,E1 58.329} C_DIS
LIN {X 0.014,Y -267.154,Z 1876.311,A 0.000,B 0.000,C 90.000,E1 55.928} C_DIS
LIN {X -0.011,Y -257.555,Z 1876.297,A 0.000,B 0.000,C 90.000,E1 53.463} C_DIS
LIN {X 0.055,Y -247.950,Z 1876.283,A 0.000,B 0.000,C 90.000,E1 50.928} C_DIS
LIN {X 0.015,Y -237.110,Z 1876.267,A 0.000,B 0.000,C 90.000,E1 48.000} C_DIS
LIN {X 0.107,Y -225.354,Z 1876.248,A 0.000,B 0.000,C 90.000,E1 44.595} C_DIS
LIN {X 0.033,Y -214.198,Z 1876.229,A 0.000,B 0.000,C 90.000,E1 41.148} C_DIS
LIN {X 0.088,Y -206.181,Z 1876.213,A 0.000,B 0.000,C 90.000,E1 38.382} C_DIS
LIN {X -0.070,Y -197.862,Z 1876.196,A 0.000,B 0.000,C 90.000,E1 35.231} C_DIS
LIN {X 0.007,Y -190.278,Z 1876.177,A 0.000,B 0.000,C 90.000,E1 31.957} C_DIS
LIN {X 0.117,Y -183.438,Z 1876.159,A 0.000,B 0.000,C 90.000,E1 28.615} C_DIS
LIN {X 0.030,Y -177.261,Z 1876.141,A 0.000,B 0.000,C 90.000,E1 25.283} C_DIS
LIN {X -0.029,Y -171.924,Z 1876.122,A 0.000,B 0.000,C 90.000,E1 21.897} C_DIS
LIN {X 0.067,Y -167.352,Z 1876.102,A 0.000,B 0.000,C 90.000,E1 18.417} C_DIS
LIN {X 0.006,Y -163.601,Z 1876.083,A 0.000,B 0.000,C 90.000,E1 14.954} C_DIS
LIN {X 0.034,Y -159.785,Z 1876.059,A 0.000,B 0.000,C 90.000,E1 10.546} C_DIS
LIN {X -0.061,Y -157.124,Z 1876.034,A 0.000,B 0.000,C 90.000,E1 6.144} C_DIS
LIN {X 0.000,Y -154.786,Z 1876.000,A 0.000,B 0.000,C 90.000,E1 360.000} C_DIS
LIN {X -0.018,Y -154.043,Z 1875.948,A 0.000,B 0.000,C 90.000,E1 350.557} C_DIS
LIN {X -0.018,Y -156.071,Z 1875.908,A 0.000,B 0.000,C 90.000,E1 343.378} C_DIS
LIN {X 0.031,Y -157.608,Z 1875.891,A 0.000,B 0.000,C 90.000,E1 340.315} C_DIS
LIN {X 0.014,Y -172.425,Z 1875.891,A 0.000,B 0.000,C 90.000,E1 340.315} C_DIS
LIN {X 0.012,Y -172.844,Z 1875.891,A 0.000,B 0.000,C 90.000,E1 340.296} C_DIS
LIN {X 0.016,Y -173.845,Z 1875.890,A 0.000,B 0.000,C 90.000,E1 340.188} C_DIS
LIN {X -0.028,Y -175.720,Z 1875.888,A 0.000,B 0.000,C 90.000,E1 339.806} C_DIS
LIN {X -0.044,Y -178.203,Z 1875.883,A 0.000,B 0.000,C 90.000,E1 338.954} C_DIS
LIN {X -0.041,Y -180.077,Z 1875.878,A 0.000,B 0.000,C 90.000,E1 338.103} C_DIS
LIN {X -0.041,Y -183.187,Z 1875.869,A 0.000,B 0.000,C 90.000,E1 336.410} C_DIS
LIN {X -0.049,Y -187.178,Z 1875.855,A 0.000,B 0.000,C 90.000,E1 333.896} C_DIS
LIN {X 0.011,Y -190.788,Z 1875.841,A 0.000,B 0.000,C 90.000,E1 331.385} C_DIS
LIN {X -0.009,Y -194.140,Z 1875.827,A 0.000,B 0.000,C 90.000,E1 328.918} C_DIS
LIN {X -0.095,Y -198.380,Z 1875.809,A 0.000,B 0.000,C 90.000,E1 325.674} C_DIS
LIN {X 0.045,Y -202.508,Z 1875.791,A 0.000,B 0.000,C 90.000,E1 322.396} C_DIS
LIN {X -0.006,Y -207.767,Z 1875.769,A 0.000,B 0.000,C 90.000,E1 318.405} C_DIS
LIN {X -0.044,Y -212.608,Z 1875.751,A 0.000,B 0.000,C 90.000,E1 315.243} C_DIS
LIN {X 0.086,Y -217.136,Z 1875.738,A 0.000,B 0.000,C 90.000,E1 312.852} C_DIS
LIN {X 0.022,Y -220.787,Z 1875.729,A 0.000,B 0.000,C 90.000,E1 311.310} C_DIS
LIN {X -0.068,Y -224.079,Z 1875.723,A 0.000,B 0.000,C 90.000,E1 310.172} C_DIS
LIN {X -0.010,Y -229.258,Z 1875.715,A 0.000,B 0.000,C 90.000,E1 308.624} C_DIS
LIN {X 0.117,Y -235.221,Z 1875.706,A 0.000,B 0.000,C 90.000,E1 307.076} C_DIS
LIN {X 0.010,Y -243.560,Z 1875.696,A 0.000,B 0.000,C 90.000,E1 305.231} C_DIS
LIN {X -0.031,Y -254.611,Z 1875.683,A 0.000,B 0.000,C 90.000,E1 303.038} C_DIS
LIN {X -0.116,Y -264.846,Z 1875.673,A 0.000,B 0.000,C 90.000,E1 301.258} C_DIS
LIN {X 0.159,Y -280.299,Z 1875.660,A 0.000,B 0.000,C 90.000,E1 298.743} C_DIS
LIN {X -0.097,Y -293.956,Z 1875.648,A 0.000,B 0.000,C 90.000,E1 296.744} C_DIS
LIN {X 0.040,Y -307.452,Z 1875.637,A 0.000,B 0.000,C 90.000,E1 294.719} C_DIS
LIN {X 0.110,Y -318.621,Z 1875.628,A 0.000,B 0.000,C 90.000,E1 293.078} C_DIS
LIN {X 0.065,Y -331.712,Z 1875.618,A 0.000,B 0.000,C 90.000,E1 291.173} C_DIS
LIN {X -0.024,Y -337.948,Z 1875.612,A 0.000,B 0.000,C 90.000,E1 290.248} C_DIS
LIN {X -0.055,Y -343.783,Z 1875.607,A 0.000,B 0.000,C 90.000,E1 289.322} C_DIS
LIN {X -0.154,Y -349.217,Z 1875.602,A 0.000,B 0.000,C 90.000,E1 288.417} C_DIS
LIN {X 0.138,Y -354.165,Z 1875.597,A 0.000,B 0.000,C 90.000,E1 287.457} C_DIS
LIN {X 0.035,Y -358.545,Z 1875.592,A 0.000,B 0.000,C 90.000,E1 286.567} C_DIS
LIN {X 0.079,Y -362.244,Z 1875.587,A 0.000,B 0.000,C 90.000,E1 285.662} C_DIS
LIN {X 0.054,Y -365.332,Z 1875.582,A 0.000,B 0.000,C 90.000,E1 284.773} C_DIS
LIN {X -0.012,Y -366.990,Z 1875.579,A 0.000,B 0.000,C 90.000,E1 284.189} C_DIS
LIN {X 0.025,Y -368.299,Z 1875.576,A 0.000,B 0.000,C 90.000,E1 283.592} C_DIS
LIN {X -0.015,Y -369.191,Z 1875.572,A 0.000,B 0.000,C 90.000,E1 283.008} C_DIS
LIN {X 0.033,Y -369.728,Z 1875.569,A 0.000,B 0.000,C 90.000,E1 282.411} C_DIS
LIN {X 0.007,Y -369.781,Z 1875.566,A 0.000,B 0.000,C 90.000,E1 281.827} C_DIS
LIN {X -0.017,Y -369.534,Z 1875.563,A 0.000,B 0.000,C 90.000,E1 281.243} C_DIS
LIN {X -0.039,Y -368.867,Z 1875.559,A 0.000,B 0.000,C 90.000,E1 280.658} C_DIS
LIN {X -0.064,Y -367.782,Z 1875.556,A 0.000,B 0.000,C 90.000,E1 280.074} C_DIS
LIN {X -0.155,Y -366.360,Z 1875.553,A 0.000,B 0.000,C 90.000,E1 279.500} C_DIS
LIN {X 0.171,Y -364.620,Z 1875.549,A 0.000,B 0.000,C 90.000,E1 278.859} C_DIS
LIN {X 0.042,Y -361.518,Z 1875.544,A 0.000,B 0.000,C 90.000,E1 277.992} C_DIS
LIN {X -0.112,Y -357.739,Z 1875.539,A 0.000,B 0.000,C 90.000,E1 277.125} C_DIS
LIN {X 0.145,Y -354.745,Z 1875.536,A 0.000,B 0.000,C 90.000,E1 276.486} C_DIS
LIN {X -0.010,Y -351.269,Z 1875.533,A 0.000,B 0.000,C 90.000,E1 275.910} C_DIS
LIN {X 0.164,Y -347.199,Z 1875.529,A 0.000,B 0.000,C 90.000,E1 275.277} C_DIS
LIN {X -0.029,Y -342.555,Z 1875.526,A 0.000,B 0.000,C 90.000,E1 274.702} C_DIS
LIN {X 0.068,Y -337.268,Z 1875.523,A 0.000,B 0.000,C 90.000,E1 274.073} C_DIS
LIN {X -0.039,Y -331.499,Z 1875.519,A 0.000,B 0.000,C 90.000,E1 273.498} C_DIS
LIN {X 0.062,Y -325.355,Z 1875.516,A 0.000,B 0.000,C 90.000,E1 272.922} C_DIS
LIN {X 0.115,Y -318.940,Z 1875.514,A 0.000,B 0.000,C 90.000,E1 272.407} C_DIS
LIN {X -0.157,Y -312.330,Z 1875.511,A 0.000,B 0.000,C 90.000,E1 272.007} C_DIS
LIN {X -0.090,Y -305.446,Z 1875.509,A 0.000,B 0.000,C 90.000,E1 271.604} C_DIS
LIN {X -0.043,Y -298.252,Z 1875.507,A 0.000,B 0.000,C 90.000,E1 271.260} C_DIS
LIN {X 0.029,Y -290.557,Z 1875.505,A 0.000,B 0.000,C 90.000,E1 270.974} C_DIS
LIN {X 0.123,Y -282.781,Z 1875.504,A 0.000,B 0.000,C 90.000,E1 270.745} C_DIS
LIN {X -0.017,Y -264.552,Z 1875.502,A 0.000,B 0.000,C 90.000,E1 270.401} C_DIS
LIN {X -0.031,Y -246.029,Z 1875.500,A 0.000,B 0.000,C 90.000,E1 270.057} C_DIS
LIN {X -0.102,Y -236.938,Z 1875.500,A 0.000,B 0.000,C 90.000,E1 269.943} C_DIS
LIN {X -0.019,Y -224.336,Z 1875.499,A 0.000,B 0.000,C 90.000,E1 269.828} C_DIS
LIN {X -0.038,Y -181.522,Z 1875.499,A 0.000,B 0.000,C 90.000,E1 269.828} C_DIS
LIN {X 0.063,Y -180.901,Z 1875.474,A 0.000,B 0.000,C 90.000,E1 265.241} C_DIS
LIN {X 0.013,Y -180.227,Z 1875.464,A 0.000,B 0.000,C 90.000,E1 263.571} C_DIS
LIN {X -0.034,Y -179.040,Z 1875.446,A 0.000,B 0.000,C 90.000,E1 260.208} C_DIS
LIN {X 0.029,Y -178.708,Z 1875.441,A 0.000,B 0.000,C 90.000,E1 259.342} C_DIS
LIN {X -0.031,Y -175.757,Z 1875.413,A 0.000,B 0.000,C 90.000,E1 254.267} C_DIS
LIN {X -0.028,Y -171.940,Z 1875.384,A 0.000,B 0.000,C 90.000,E1 249.135} C_DIS
LIN {X -0.052,Y -171.324,Z 1875.379,A 0.000,B 0.000,C 90.000,E1 248.284} C_DIS
LIN {X 0.001,Y -167.580,Z 1875.355,A 0.000,B 0.000,C 90.000,E1 243.948} C_DIS
LIN {X -0.060,Y -166.214,Z 1875.346,A 0.000,B 0.000,C 90.000,E1 242.231} C_DIS
LIN {X -0.071,Y -162.978,Z 1875.326,A 0.000,B 0.000,C 90.000,E1 238.742} C_DIS
LIN {X -0.024,Y -160.891,Z 1875.312,A 0.000,B 0.000,C 90.000,E1 236.087} C_DIS
LIN {X -0.045,Y -157.661,Z 1875.292,A 0.000,B 0.000,C 90.000,E1 232.557} C_DIS
LIN {X 0.013,Y -155.698,Z 1875.277,A 0.000,B 0.000,C 90.000,E1 229.865} C_DIS
LIN {X -0.051,Y -151.961,Z 1875.252,A 0.000,B 0.000,C 90.000,E1 225.405} C_DIS
LIN {X -0.035,Y -150.203,Z 1875.237,A 0.000,B 0.000,C 90.000,E1 222.690} C_DIS
LIN {X 0.096,Y -146.971,Z 1875.212,A 0.000,B 0.000,C 90.000,E1 218.096} C_DIS
LIN {X -0.001,Y -145.558,Z 1875.197,A 0.000,B 0.000,C 90.000,E1 215.391} C_DIS
LIN {X -0.001,Y -142.951,Z 1875.171,A 0.000,B 0.000,C 90.000,E1 210.797} C_DIS
LIN {X -0.070,Y -141.577,Z 1875.151,A 0.000,B 0.000,C 90.000,E1 207.129} C_DIS
LIN {X -0.023,Y -139.414,Z 1875.115,A 0.000,B 0.000,C 90.000,E1 200.610} C_DIS
LIN {X 0.029,Y -139.138,Z 1875.104,A 0.000,B 0.000,C 90.000,E1 198.725} C_DIS
LIN {X 0.056,Y -138.349,Z 1875.057,A 0.000,B 0.000,C 90.000,E1 190.310} C_DIS
LIN {X 0.044,Y -139.493,Z 1875.005,A 0.000,B 0.000,C 90.000,E1 180.974} C_DIS
LIN {X -0.015,Y -141.106,Z 1874.974,A 0.000,B 0.000,C 90.000,E1 175.412} C_DIS
LIN {X -0.061,Y -142.485,Z 1874.959,A 0.000,B 0.000,C 90.000,E1 172.648} C_DIS
LIN {X 0.026,Y -144.736,Z 1874.933,A 0.000,B 0.000,C 90.000,E1 167.993} C_DIS
LIN {X -0.023,Y -147.341,Z 1874.913,A 0.000,B 0.000,C 90.000,E1 164.338} C_DIS
LIN {X 0.042,Y -150.665,Z 1874.888,A 0.000,B 0.000,C 90.000,E1 159.752} C_DIS
LIN {X -0.077,Y -154.144,Z 1874.867,A 0.000,B 0.000,C 90.000,E1 156.177} C_DIS
LIN {X 0.058,Y -157.574,Z 1874.848,A 0.000,B 0.000,C 90.000,E1 152.538} C_DIS
LIN {X 0.009,Y -161.819,Z 1874.828,A 0.000,B 0.000,C 90.000,E1 148.997} C_DIS
LIN {X 0.028,Y -166.009,Z 1874.808,A 0.000,B 0.000,C 90.000,E1 145.468} C_DIS
LIN {X 0.021,Y -171.009,Z 1874.789,A 0.000,B 0.000,C 90.000,E1 141.984} C_DIS
LIN {X 0.052,Y -175.879,Z 1874.770,A 0.000,B 0.000,C 90.000,E1 138.528} C_DIS
LIN {X -0.071,Y -181.484,Z 1874.751,A 0.000,B 0.000,C 90.000,E1 135.162} C_DIS
LIN {X 0.065,Y -186.998,Z 1874.732,A 0.000,B 0.000,C 90.000,E1 131.757} C_DIS
LIN {X 0.067,Y -190.115,Z 1874.723,A 0.000,B 0.000,C 90.000,E1 130.092} C_DIS
LIN {X 0.086,Y -195.886,Z 1874.704,A 0.000,B 0.000,C 90.000,E1 126.790} C_DIS
LIN {X -0.123,Y -200.718,Z 1874.691,A 0.000,B 0.000,C 90.000,E1 124.405} C_DIS
LIN {X 0.069,Y -206.605,Z 1874.673,A 0.000,B 0.000,C 90.000,E1 121.131} C_DIS
LIN {X 0.061,Y -209.899,Z 1874.664,A 0.000,B 0.000,C 90.000,E1 119.539} C_DIS
LIN {X 0.092,Y -217.255,Z 1874.642,A 0.000,B 0.000,C 90.000,E1 115.591} C_DIS
LIN {X 0.045,Y -218.880,Z 1874.638,A 0.000,B 0.000,C 90.000,E1 114.823} C_DIS
LIN {X 0.017,Y -224.102,Z 1874.621,A 0.000,B 0.000,C 90.000,E1 111.844} C_DIS
LIN {X -0.016,Y -283.635,Z 1874.621,A 0.000,B 0.000,C 90.000,E1 111.844} C_DIS
LIN {X 0.109,Y -287.419,Z 1874.621,A 0.000,B 0.000,C 90.000,E1 111.716} C_DIS
LIN {X -0.027,Y -290.664,Z 1874.620,A 0.000,B 0.000,C 90.000,E1 111.535} C_DIS
LIN {X -0.062,Y -294.304,Z 1874.617,A 0.000,B 0.000,C 90.000,E1 111.153} C_DIS
LIN {X -0.022,Y -296.265,Z 1874.616,A 0.000,B 0.000,C 90.000,E1 110.844} C_DIS
LIN {X 0.054,Y -309.302,Z 1874.603,A 0.000,B 0.000,C 90.000,E1 108.544} C_DIS
END
